gfCNCPoint1[24009] = {X 25.7631, Y 5.7856, Z -2.1667, A 0.000, B 0.000, C 0.000 }
gfCNCPoint1[24010] = {X 27.5759, Y 7.0515, Z -2.1667, A 0.000, B 0.000, C 0.000 }
gfCNCPoint1[24011] = {X 28.5579, Y 7.8754, Z -2.1667, A 0.000, B 0.000, C 0.000 }
gfCNCPoint1[24012] = {X 29.4785, Y 8.7676, Z -2.1667, A 0.000, B 0.000, C 0.000 }
gfCNCPoint1[24013] = {X 30.6864, Y 10.1626, Z -2.1667, A 0.000, B 0.000, C 0.000 }
gfCNCPoint1[24014] = {X 31.7443, Y 11.6745, Z -2.1667, A 0.000, B 0.000, C 0.000 }
gfCNCPoint1[24015] = {X 32.6409, Y 13.2874, Z -2.1667, A 0.000, B 0.000, C 0.000 }
gfCNCPoint1[24016] = {X 33.3666, Y 14.9840, Z -2.1667, A 0.000, B 0.000, C 0.000 }
gfCNCPoint1[24017] = {X 33.9177, Y 16.8152, Z -2.1667, A 0.000, B 0.000, C 0.000 }
gfCNCPoint1[24018] = {X 34.2900, Y 18.6910, Z -2.1667, A 0.000, B 0.000, C 0.000 }
gfCNCPoint1[24019] = {X 34.4801, Y 20.5940, Z -2.1667, A 0.000, B 0.000, C 0.000 }
gfCNCPoint1[24020] = {X 34.4863, Y 22.5063, Z -2.1667, A 0.000, B 0.000, C 0.000 }
gfCNCPoint1[24021] = {X 34.3084, Y 24.4105, Z -2.1667, A 0.000, B 0.000, C 0.000 }
gfCNCPoint1[24022] = {X 33.9482, Y 26.2886, Z -2.1667, A 0.000, B 0.000, C 0.000 }
gfCNCPoint1[24023] = {X 33.4648, Y 27.9398, Z -2.1667, A 0.000, B 0.000, C 0.000 }
gfCNCPoint1[24024] = {X 32.8126, Y 29.5319, Z -2.1667, A 0.000, B 0.000, C 0.000 }
gfCNCPoint1[24025] = {X 31.9989, Y 31.0478, Z -2.1667, A 0.000, B 0.000, C 0.000 }
gfCNCPoint1[24026] = {X 32.1285, Y 31.2838, Z -2.1667, A 0.000, B 0.000, C 0.000 }
gfCNCPoint1[24027] = {X 32.2512, Y 31.5235, Z -2.1667, A 0.000, B 0.000, C 0.000 }
gfCNCPoint1[24028] = {X 35.3025, Y 37.8269, Z -2.1667, A 0.000, B 0.000, C 0.000 }
gfCNCPoint1[24029] = {X 35.7263, Y 38.8573, Z -2.1667, A 0.000, B 0.000, C 0.000 }
gfCNCPoint1[24030] = {X 36.0224, Y 39.9313, Z -2.1667, A 0.000, B 0.000, C 0.000 }
gfCNCPoint1[24031] = {X 36.1865, Y 41.0332, Z -2.1667, A 0.000, B 0.000, C 0.000 }
gfCNCPoint1[24032] = {X 36.2163, Y 42.1469, Z -2.1667, A 0.000, B 0.000, C 0.000 }
gfCNCPoint1[24033] = {X 36.6306, Y 41.4259, Z -2.1667, A 0.000, B 0.000, C 0.000 }
gfCNCPoint1[24034] = {X 37.1613, Y 40.7857, Z -2.1667, A 0.000, B 0.000, C 0.000 }
gfCNCPoint1[24035] = {X 37.7930, Y 40.2449, Z -2.1667, A 0.000, B 0.000, C 0.000 }
gfCNCPoint1[24036] = {X 38.5073, Y 39.8191, Z -2.1667, A 0.000, B 0.000, C 0.000 }
gfCNCPoint1[24037] = {X 39.0456, Y 38.5336, Z -2.1667, A 0.000, B 0.000, C 0.000 }
gfCNCPoint1[24038] = {X 39.5416, Y 37.2312, Z -2.1667, A 0.000, B 0.000, C 0.000 }
gfCNCPoint1[24039] = {X 47.6703, Y 15.4045, Z -2.1667, A 0.000, B 0.000, C 0.000 }
gfCNCPoint1[24040] = {X 47.3200, Y 14.6512, Z -2.1667, A 0.000, B 0.000, C 0.000 }
gfCNCPoint1[24041] = {X 47.1026, Y 13.8493, Z -2.1667, A 0.000, B 0.000, C 0.000 }
gfCNCPoint1[24042] = {X 47.0244, Y 13.0222, Z -2.1667, A 0.000, B 0.000, C 0.000 }
gfCNCPoint1[24043] = {X 47.0242, Y 12.1868, Z -2.1667, A 0.000, B 0.000, C 0.000 }
gfCNCPoint1[24044] = {X 47.0722, Y 11.5041, Z -2.1667, A 0.000, B 0.000, C 0.000 }
gfCNCPoint1[24045] = {X 47.2152, Y 10.8349, Z -2.1667, A 0.000, B 0.000, C 0.000 }
gfCNCPoint1[24046] = {X 42.6031, Y 9.5051, Z -2.1667, A 0.000, B 0.000, C 0.000 }
gfCNCPoint1[24047] = {X 36.0439, Y 9.5051, Z -2.1667, A 0.000, B 0.000, C 0.000 }
gfCNCPoint1[24048] = {X 37.0532, Y 11.3861, Z -2.1667, A 0.000, B 0.000, C 0.000 }
gfCNCPoint1[24049] = {X 37.8813, Y 13.3537, Z -2.1667, A 0.000, B 0.000, C 0.000 }
gfCNCPoint1[24050] = {X 38.5455, Y 15.5364, Z -2.1667, A 0.000, B 0.000, C 0.000 }
gfCNCPoint1[24051] = {X 39.0050, Y 17.7712, Z -2.1667, A 0.000, B 0.000, C 0.000 }
gfCNCPoint1[24052] = {X 39.2560, Y 20.0389, Z -2.1667, A 0.000, B 0.000, C 0.000 }
gfCNCPoint1[24053] = {X 39.2962, Y 22.3201, Z -2.1667, A 0.000, B 0.000, C 0.000 }
gfCNCPoint1[24054] = {X 39.1255, Y 24.5952, Z -2.1667, A 0.000, B 0.000, C 0.000 }
gfCNCPoint1[24055] = {X 42.5394, Y 15.4281, Z -2.1667, A 0.000, B 0.000, C 0.000 }
gfCNCPoint1[24056] = {X 42.3081, Y 14.2498, Z -2.1667, A 0.000, B 0.000, C 0.000 }
gfCNCPoint1[24057] = {X 42.2245, Y 13.0519, Z -2.1667, A 0.000, B 0.000, C 0.000 }
gfCNCPoint1[24058] = {X 42.2242, Y 12.1868, Z -2.1667, A 0.000, B 0.000, C 0.000 }
gfCNCPoint1[24059] = {X 42.3194, Y 10.8326, Z -2.1667, A 0.000, B 0.000, C 0.000 }
gfCNCPoint1[24060] = {X 42.6031, Y 9.5051, Z -2.1667, A 0.000, B 0.000, C 0.000 }
gfCNCPoint1[24061] = {X 44.9092, Y 10.1700, Z -2.1667, A 0.000, B 0.000, C 0.000 }
gfCNCPoint1[24062] = {X 45.3323, Y 9.0551, Z -2.1667, A 0.000, B 0.000, C 0.000 }
gfCNCPoint1[24063] = {X 45.9317, Y 8.0242, Z -2.1667, A 0.000, B 0.000, C 0.000 }
gfCNCPoint1[24064] = {X 46.6913, Y 7.1051, Z -2.1667, A 0.000, B 0.000, C 0.000 }
gfCNCPoint1[24065] = {X 31.2094, Y 7.1051, Z -2.1667, A 0.000, B 0.000, C 0.000 }
gfCNCPoint1[24066] = {X 32.2249, Y 8.2452, Z -2.1667, A 0.000, B 0.000, C 0.000 }
gfCNCPoint1[24067] = {X 33.1518, Y 9.4585, Z -2.1667, A 0.000, B 0.000, C 0.000 }
gfCNCPoint1[24068] = {X 33.9848, Y 10.7380, Z -2.1667, A 0.000, B 0.000, C 0.000 }
gfCNCPoint1[24069] = {X 34.8849, Y 12.4149, Z -2.1667, A 0.000, B 0.000, C 0.000 }
gfCNCPoint1[24070] = {X 35.6240, Y 14.1688, Z -2.1667, A 0.000, B 0.000, C 0.000 }
gfCNCPoint1[24071] = {X 36.2218, Y 16.1371, Z -2.1667, A 0.000, B 0.000, C 0.000 }
gfCNCPoint1[24072] = {X 36.6354, Y 18.1522, Z -2.1667, A 0.000, B 0.000, C 0.000 }
gfCNCPoint1[24073] = {X 36.8612, Y 20.1969, Z -2.1667, A 0.000, B 0.000, C 0.000 }
gfCNCPoint1[24074] = {X 36.8971, Y 22.2537, Z -2.1667, A 0.000, B 0.000, C 0.000 }
gfCNCPoint1[24075] = {X 36.7431, Y 24.3050, Z -2.1667, A 0.000, B 0.000, C 0.000 }
gfCNCPoint1[24076] = {X 36.5495, Y 25.5833, Z -2.1667, A 0.000, B 0.000, C 0.000 }
gfCNCPoint1[24077] = {X 36.2821, Y 26.8481, Z -2.1667, A 0.000, B 0.000, C 0.000 }
gfCNCPoint1[24078] = {X 35.8735, Y 28.3068, Z -2.1667, A 0.000, B 0.000, C 0.000 }
gfCNCPoint1[24079] = {X 35.3497, Y 29.7282, Z -2.1667, A 0.000, B 0.000, C 0.000 }
gfCNCPoint1[24080] = {X 34.7142, Y 31.1033, Z -2.1667, A 0.000, B 0.000, C 0.000 }
gfCNCPoint1[24081] = {X 37.2850, Y 36.4140, Z -2.1667, A 0.000, B 0.000, C 0.000 }
gfCNCPoint1[24082] = {X 45.0744, Y 15.4982, Z -2.1667, A 0.000, B 0.000, C 0.000 }
gfCNCPoint1[24083] = {X 44.7426, Y 14.2853, Z -2.1667, A 0.000, B 0.000, C 0.000 }
gfCNCPoint1[24084] = {X 44.6244, Y 13.0334, Z -2.1667, A 0.000, B 0.000, C 0.000 }
gfCNCPoint1[24085] = {X 44.6242, Y 12.1868, Z -2.1667, A 0.000, B 0.000, C 0.000 }
gfCNCPoint1[24086] = {X 44.6958, Y 11.1684, Z -2.1667, A 0.000, B 0.000, C 0.000 }
gfCNCPoint1[24087] = {X 44.9092, Y 10.1700, Z -2.1667, A 0.000, B 0.000, C 0.000 }
gfCNCPoint1[24088] = {X 47.2152, Y 10.8349, Z -2.1667, A 0.000, B 0.000, C 0.000 }
gfCNCPoint1[24089] = {X 47.4988, Y 10.0875, Z -2.1667, A 0.000, B 0.000, C 0.000 }
gfCNCPoint1[24090] = {X 47.9006, Y 9.3965, Z -2.1667, A 0.000, B 0.000, C 0.000 }
gfCNCPoint1[24091] = {X 48.4099, Y 8.7804, Z -2.1667, A 0.000, B 0.000, C 0.000 }
gfCNCPoint1[24092] = {X 49.1544, Y 8.1553, Z -2.1667, A 0.000, B 0.000, C 0.000 }
gfCNCPoint1[24093] = {X 50.0080, Y 7.6903, Z -2.1667, A 0.000, B 0.000, C 0.000 }
gfCNCPoint1[24094] = {X 50.9369, Y 7.4036, Z -2.1667, A 0.000, B 0.000, C 0.000 }
gfCNCPoint1[24095] = {X 51.9042, Y 7.3068, Z -2.1667, A 0.000, B 0.000, C 0.000 }
gfCNCPoint1[24096] = {X 59.6221, Y 7.3068, Z -2.1667, A 0.000, B 0.000, C 0.000 }
gfCNCPoint1[24097] = {X 60.5894, Y 7.4036, Z -2.1667, A 0.000, B 0.000, C 0.000 }
gfCNCPoint1[24098] = {X 61.5183, Y 7.6903, Z -2.1667, A 0.000, B 0.000, C 0.000 }
gfCNCPoint1[24099] = {X 62.3720, Y 8.1553, Z -2.1667, A 0.000, B 0.000, C 0.000 }
gfCNCPoint1[24100] = {X 63.1165, Y 8.7804, Z -2.1667, A 0.000, B 0.000, C 0.000 }
gfCNCPoint1[24101] = {X 63.7054, Y 9.5145, Z -2.1667, A 0.000, B 0.000, C 0.000 }
gfCNCPoint1[24102] = {X 64.1425, Y 10.3481, Z -2.1667, A 0.000, B 0.000, C 0.000 }
gfCNCPoint1[24103] = {X 64.4114, Y 11.2500, Z -2.1667, A 0.000, B 0.000, C 0.000 }
gfCNCPoint1[24104] = {X 64.5021, Y 12.1868, Z -2.1667, A 0.000, B 0.000, C 0.000 }
gfCNCPoint1[24105] = {X 64.5019, Y 13.0237, Z -2.1667, A 0.000, B 0.000, C 0.000 }
gfCNCPoint1[24106] = {X 64.4204, Y 13.8671, Z -2.1667, A 0.000, B 0.000, C 0.000 }
gfCNCPoint1[24107] = {X 64.1943, Y 14.6838, Z -2.1667, A 0.000, B 0.000, C 0.000 }
gfCNCPoint1[24108] = {X 63.8303, Y 15.4490, Z -2.1667, A 0.000, B 0.000, C 0.000 }
gfCNCPoint1[24109] = {X 63.9941, Y 15.8770, Z -2.1667, A 0.000, B 0.000, C 0.000 }
gfCNCPoint1[24110] = {X 72.9532, Y 39.8573, Z -2.1667, A 0.000, B 0.000, C 0.000 }
gfCNCPoint1[24111] = {X 73.8435, Y 40.4391, Z -2.1667, A 0.000, B 0.000, C 0.000 }
gfCNCPoint1[24112] = {X 74.5866, Y 41.2001, Z -2.1667, A 0.000, B 0.000, C 0.000 }
gfCNCPoint1[24113] = {X 75.1472, Y 42.1040, Z -2.1667, A 0.000, B 0.000, C 0.000 }
gfCNCPoint1[24114] = {X 75.4987, Y 43.1079, Z -2.1667, A 0.000, B 0.000, C 0.000 }
gfCNCPoint1[24115] = {X 75.6243, Y 44.1640, Z -2.1667, A 0.000, B 0.000, C 0.000 }
gfCNCPoint1[24116] = {X 75.6245, Y 45.0000, Z -2.1667, A 0.000, B 0.000, C 0.000 }
gfCNCPoint1[24117] = {X 75.5307, Y 45.9520, Z -2.1667, A 0.000, B 0.000, C 0.000 }
gfCNCPoint1[24118] = {X 75.2530, Y 46.8675, Z -2.1667, A 0.000, B 0.000, C 0.000 }
gfCNCPoint1[24119] = {X 74.8020, Y 47.7112, Z -2.1667, A 0.000, B 0.000, C 0.000 }
gfCNCPoint1[24120] = {X 74.1951, Y 48.4507, Z -2.1667, A 0.000, B 0.000, C 0.000 }
gfCNCPoint1[24121] = {X 73.4556, Y 49.0576, Z -2.1667, A 0.000, B 0.000, C 0.000 }
gfCNCPoint1[24122] = {X 72.6120, Y 49.5085, Z -2.1667, A 0.000, B 0.000, C 0.000 }
gfCNCPoint1[24123] = {X 71.6965, Y 49.7862, Z -2.1667, A 0.000, B 0.000, C 0.000 }
gfCNCPoint1[24124] = {X 70.7445, Y 49.8800, Z -2.1667, A 0.000, B 0.000, C 0.000 }
gfCNCPoint1[24125] = {X 64.1851, Y 49.8800, Z -2.1667, A 0.000, B 0.000, C 0.000 }
gfCNCPoint1[24126] = {X 63.2331, Y 49.7862, Z -2.1667, A 0.000, B 0.000, C 0.000 }
gfCNCPoint1[24127] = {X 62.3176, Y 49.5085, Z -2.1667, A 0.000, B 0.000, C 0.000 }
gfCNCPoint1[24128] = {X 61.4740, Y 49.0576, Z -2.1667, A 0.000, B 0.000, C 0.000 }
gfCNCPoint1[24129] = {X 60.7345, Y 48.4507, Z -2.1667, A 0.000, B 0.000, C 0.000 }
gfCNCPoint1[24130] = {X 60.1276, Y 47.7112, Z -2.1667, A 0.000, B 0.000, C 0.000 }
gfCNCPoint1[24131] = {X 59.6766, Y 46.8675, Z -2.1667, A 0.000, B 0.000, C 0.000 }
gfCNCPoint1[24132] = {X 59.3989, Y 45.9520, Z -2.1667, A 0.000, B 0.000, C 0.000 }
gfCNCPoint1[24133] = {X 59.3051, Y 45.0000, Z -2.1667, A 0.000, B 0.000, C 0.000 }
gfCNCPoint1[24134] = {X 59.3052, Y 44.2029, Z -2.1667, A 0.000, B 0.000, C 0.000 }
gfCNCPoint1[24135] = {X 59.3848, Y 43.3308, Z -2.1667, A 0.000, B 0.000, C 0.000 }
gfCNCPoint1[24136] = {X 59.6190, Y 42.4870, Z -2.1667, A 0.000, B 0.000, C 0.000 }
gfCNCPoint1[24137] = {X 60.0003, Y 41.6986, Z -2.1667, A 0.000, B 0.000, C 0.000 }
gfCNCPoint1[24138] = {X 59.6160, Y 40.6492, Z -2.1667, A 0.000, B 0.000, C 0.000 }
gfCNCPoint1[24139] = {X 52.4655, Y 40.6492, Z -2.1667, A 0.000, B 0.000, C 0.000 }
gfCNCPoint1[24140] = {X 51.9464, Y 42.0438, Z -2.1667, A 0.000, B 0.000, C 0.000 }
gfCNCPoint1[24141] = {X 52.2214, Y 42.7234, Z -2.1667, A 0.000, B 0.000, C 0.000 }
gfCNCPoint1[24142] = {X 52.3914, Y 43.4366, Z -2.1667, A 0.000, B 0.000, C 0.000 }
gfCNCPoint1[24143] = {X 52.4528, Y 44.1672, Z -2.1667, A 0.000, B 0.000, C 0.000 }
gfCNCPoint1[24144] = {X 52.4529, Y 45.0000, Z -2.1667, A 0.000, B 0.000, C 0.000 }
gfCNCPoint1[24145] = {X 52.3592, Y 45.9520, Z -2.1667, A 0.000, B 0.000, C 0.000 }
gfCNCPoint1[24146] = {X 52.0815, Y 46.8675, Z -2.1667, A 0.000, B 0.000, C 0.000 }
gfCNCPoint1[24147] = {X 51.6305, Y 47.7112, Z -2.1667, A 0.000, B 0.000, C 0.000 }
gfCNCPoint1[24148] = {X 51.0236, Y 48.4507, Z -2.1667, A 0.000, B 0.000, C 0.000 }
gfCNCPoint1[24149] = {X 50.2841, Y 49.0576, Z -2.1667, A 0.000, B 0.000, C 0.000 }
gfCNCPoint1[24150] = {X 49.4404, Y 49.5085, Z -2.1667, A 0.000, B 0.000, C 0.000 }
gfCNCPoint1[24151] = {X 48.5250, Y 49.7862, Z -2.1667, A 0.000, B 0.000, C 0.000 }
gfCNCPoint1[24152] = {X 47.5729, Y 49.8800, Z -2.1667, A 0.000, B 0.000, C 0.000 }
gfCNCPoint1[24153] = {X 40.6393, Y 49.8800, Z -2.1667, A 0.000, B 0.000, C 0.000 }
gfCNCPoint1[24154] = {X 39.6433, Y 49.7773, Z -2.1667, A 0.000, B 0.000, C 0.000 }
gfCNCPoint1[24155] = {X 38.6892, Y 49.4734, Z -2.1667, A 0.000, B 0.000, C 0.000 }
gfCNCPoint1[24156] = {X 37.8173, Y 48.9813, Z -2.1667, A 0.000, B 0.000, C 0.000 }
gfCNCPoint1[24157] = {X 37.0641, Y 48.3215, Z -2.1667, A 0.000, B 0.000, C 0.000 }
gfCNCPoint1[24158] = {X 36.5085, Y 47.5983, Z -2.1667, A 0.000, B 0.000, C 0.000 }
gfCNCPoint1[24159] = {X 36.0972, Y 46.7843, Z -2.1667, A 0.000, B 0.000, C 0.000 }
gfCNCPoint1[24160] = {X 35.8445, Y 45.9080, Z -2.1667, A 0.000, B 0.000, C 0.000 }
gfCNCPoint1[24161] = {X 35.7593, Y 45.0000, Z -2.1667, A 0.000, B 0.000, C 0.000 }
gfCNCPoint1[24162] = {X 35.7593, Y 44.7148, Z -2.1667, A 0.000, B 0.000, C 0.000 }
gfCNCPoint1[24163] = {X 36.2393, Y 44.7148, Z -2.1667, A 0.000, B 0.000, C 0.000 }
gfCNCPoint1[24164] = {X 36.2397, Y 44.1483, Z -2.1667, A 0.000, B 0.000, C 0.000 }
gfCNCPoint1[24165] = {X 36.3681, Y 43.1519, Z -2.1667, A 0.000, B 0.000, C 0.000 }
gfCNCPoint1[24166] = {X 36.7192, Y 42.2107, Z -2.1667, A 0.000, B 0.000, C 0.000 }
gfCNCPoint1[24167] = {X 37.2745, Y 41.3736, Z -2.1667, A 0.000, B 0.000, C 0.000 }
gfCNCPoint1[24168] = {X 38.0053, Y 40.6843, Z -2.1667, A 0.000, B 0.000, C 0.000 }
gfCNCPoint1[24169] = {X 38.8734, Y 40.1787, Z -2.1667, A 0.000, B 0.000, C 0.000 }
gfCNCPoint1[24170] = {X 39.4565, Y 38.7984, Z -2.1667, A 0.000, B 0.000, C 0.000 }
gfCNCPoint1[24171] = {X 39.9914, Y 37.3987, Z -2.1667, A 0.000, B 0.000, C 0.000 }
gfCNCPoint1[24172] = {X 48.2011, Y 15.3544, Z -2.1667, A 0.000, B 0.000, C 0.000 }
gfCNCPoint1[24173] = {X 47.8187, Y 14.6115, Z -2.1667, A 0.000, B 0.000, C 0.000 }
gfCNCPoint1[24174] = {X 47.5835, Y 13.8097, Z -2.1667, A 0.000, B 0.000, C 0.000 }
gfCNCPoint1[24175] = {X 47.5042, Y 12.9779, Z -2.1667, A 0.000, B 0.000, C 0.000 }
gfCNCPoint1[24176] = {X 47.5042, Y 12.1868, Z -2.1667, A 0.000, B 0.000, C 0.000 }
gfCNCPoint1[24177] = {X 47.6145, Y 11.2077, Z -2.1667, A 0.000, B 0.000, C 0.000 }
gfCNCPoint1[24178] = {X 47.9400, Y 10.2777, Z -2.1667, A 0.000, B 0.000, C 0.000 }
gfCNCPoint1[24179] = {X 48.4642, Y 9.4435, Z -2.1667, A 0.000, B 0.000, C 0.000 }
gfCNCPoint1[24180] = {X 49.1609, Y 8.7468, Z -2.1667, A 0.000, B 0.000, C 0.000 }
gfCNCPoint1[24181] = {X 49.9951, Y 8.2226, Z -2.1667, A 0.000, B 0.000, C 0.000 }
gfCNCPoint1[24182] = {X 50.9251, Y 7.8971, Z -2.1667, A 0.000, B 0.000, C 0.000 }
gfCNCPoint1[24183] = {X 51.9042, Y 7.7868, Z -2.1667, A 0.000, B 0.000, C 0.000 }
gfCNCPoint1[24184] = {X 59.6221, Y 7.7868, Z -2.1667, A 0.000, B 0.000, C 0.000 }
gfCNCPoint1[24185] = {X 60.6012, Y 7.8971, Z -2.1667, A 0.000, B 0.000, C 0.000 }
gfCNCPoint1[24186] = {X 61.5312, Y 8.2226, Z -2.1667, A 0.000, B 0.000, C 0.000 }
gfCNCPoint1[24187] = {X 62.3655, Y 8.7468, Z -2.1667, A 0.000, B 0.000, C 0.000 }
gfCNCPoint1[24188] = {X 63.0622, Y 9.4435, Z -2.1667, A 0.000, B 0.000, C 0.000 }
gfCNCPoint1[24189] = {X 63.5864, Y 10.2777, Z -2.1667, A 0.000, B 0.000, C 0.000 }
gfCNCPoint1[24190] = {X 63.9118, Y 11.2077, Z -2.1667, A 0.000, B 0.000, C 0.000 }
gfCNCPoint1[24191] = {X 64.0221, Y 12.1868, Z -2.1667, A 0.000, B 0.000, C 0.000 }
gfCNCPoint1[24192] = {X 64.0219, Y 13.0233, Z -2.1667, A 0.000, B 0.000, C 0.000 }
gfCNCPoint1[24193] = {X 63.9336, Y 13.8564, Z -2.1667, A 0.000, B 0.000, C 0.000 }
gfCNCPoint1[24194] = {X 63.6889, Y 14.6576, Z -2.1667, A 0.000, B 0.000, C 0.000 }
gfCNCPoint1[24195] = {X 63.2969, Y 15.3980, Z -2.1667, A 0.000, B 0.000, C 0.000 }
gfCNCPoint1[24196] = {X 63.5448, Y 16.0461, Z -2.1667, A 0.000, B 0.000, C 0.000 }
gfCNCPoint1[24197] = {X 66.1094, Y 22.8602, Z -2.1667, A 0.000, B 0.000, C 0.000 }
gfCNCPoint1[24198] = {X 72.2834, Y 39.4716, Z -2.1667, A 0.000, B 0.000, C 0.000 }
gfCNCPoint1[24199] = {X 72.5762, Y 40.2082, Z -2.1667, A 0.000, B 0.000, C 0.000 }
gfCNCPoint1[24200] = {X 73.4340, Y 40.7265, Z -2.1667, A 0.000, B 0.000, C 0.000 }
gfCNCPoint1[24201] = {X 74.1523, Y 41.4256, Z -2.1667, A 0.000, B 0.000, C 0.000 }
gfCNCPoint1[24202] = {X 74.6938, Y 42.2690, Z -2.1667, A 0.000, B 0.000, C 0.000 }
gfCNCPoint1[24203] = {X 75.0303, Y 43.2131, Z -2.1667, A 0.000, B 0.000, C 0.000 }
gfCNCPoint1[24204] = {X 75.1445, Y 44.2089, Z -2.1667, A 0.000, B 0.000, C 0.000 }
gfCNCPoint1[24205] = {X 75.1445, Y 45.0000, Z -2.1667, A 0.000, B 0.000, C 0.000 }
gfCNCPoint1[24206] = {X 75.0341, Y 45.9791, Z -2.1667, A 0.000, B 0.000, C 0.000 }
gfCNCPoint1[24207] = {X 74.7087, Y 46.9091, Z -2.1667, A 0.000, B 0.000, C 0.000 }
gfCNCPoint1[24208] = {X 74.1845, Y 47.7434, Z -2.1667, A 0.000, B 0.000, C 0.000 }
gfCNCPoint1[24209] = {X 73.4878, Y 48.4401, Z -2.1667, A 0.000, B 0.000, C 0.000 }
gfCNCPoint1[24210] = {X 72.6535, Y 48.9643, Z -2.1667, A 0.000, B 0.000, C 0.000 }
gfCNCPoint1[24211] = {X 71.7236, Y 49.2897, Z -2.1667, A 0.000, B 0.000, C 0.000 }
gfCNCPoint1[24212] = {X 70.7445, Y 49.4000, Z -2.1667, A 0.000, B 0.000, C 0.000 }
gfCNCPoint1[24213] = {X 64.1851, Y 49.4000, Z -2.1667, A 0.000, B 0.000, C 0.000 }
gfCNCPoint1[24214] = {X 63.2060, Y 49.2897, Z -2.1667, A 0.000, B 0.000, C 0.000 }
gfCNCPoint1[24215] = {X 62.2760, Y 48.9643, Z -2.1667, A 0.000, B 0.000, C 0.000 }
gfCNCPoint1[24216] = {X 61.4418, Y 48.4401, Z -2.1667, A 0.000, B 0.000, C 0.000 }
gfCNCPoint1[24217] = {X 60.7451, Y 47.7434, Z -2.1667, A 0.000, B 0.000, C 0.000 }
gfCNCPoint1[24218] = {X 60.2209, Y 46.9091, Z -2.1667, A 0.000, B 0.000, C 0.000 }
gfCNCPoint1[24219] = {X 59.8955, Y 45.9791, Z -2.1667, A 0.000, B 0.000, C 0.000 }
gfCNCPoint1[24220] = {X 59.7851, Y 45.0000, Z -2.1667, A 0.000, B 0.000, C 0.000 }
gfCNCPoint1[24221] = {X 59.7856, Y 44.1483, Z -2.1667, A 0.000, B 0.000, C 0.000 }
gfCNCPoint1[24222] = {X 59.8784, Y 43.3075, Z -2.1667, A 0.000, B 0.000, C 0.000 }
gfCNCPoint1[24223] = {X 60.1305, Y 42.5001, Z -2.1667, A 0.000, B 0.000, C 0.000 }
gfCNCPoint1[24224] = {X 60.5324, Y 41.7558, Z -2.1667, A 0.000, B 0.000, C 0.000 }
gfCNCPoint1[24225] = {X 59.9515, Y 40.1692, Z -2.1667, A 0.000, B 0.000, C 0.000 }
gfCNCPoint1[24226] = {X 52.1320, Y 40.1692, Z -2.1667, A 0.000, B 0.000, C 0.000 }
gfCNCPoint1[24227] = {X 51.4219, Y 42.0768, Z -2.1667, A 0.000, B 0.000, C 0.000 }
gfCNCPoint1[24228] = {X 51.7251, Y 42.7530, Z -2.1667, A 0.000, B 0.000, C 0.000 }
gfCNCPoint1[24229] = {X 51.9105, Y 43.4705, Z -2.1667, A 0.000, B 0.000, C 0.000 }
gfCNCPoint1[24230] = {X 51.9729, Y 44.2089, Z -2.1667, A 0.000, B 0.000, C 0.000 }
gfCNCPoint1[24231] = {X 51.9729, Y 45.0000, Z -2.1667, A 0.000, B 0.000, C 0.000 }
gfCNCPoint1[24232] = {X 51.8626, Y 45.9791, Z -2.1667, A 0.000, B 0.000, C 0.000 }
gfCNCPoint1[24233] = {X 51.5372, Y 46.9091, Z -2.1667, A 0.000, B 0.000, C 0.000 }
gfCNCPoint1[24234] = {X 51.0130, Y 47.7434, Z -2.1667, A 0.000, B 0.000, C 0.000 }
gfCNCPoint1[24235] = {X 50.3163, Y 48.4401, Z -2.1667, A 0.000, B 0.000, C 0.000 }
gfCNCPoint1[24236] = {X 49.4820, Y 48.9643, Z -2.1667, A 0.000, B 0.000, C 0.000 }
gfCNCPoint1[24237] = {X 48.5520, Y 49.2897, Z -2.1667, A 0.000, B 0.000, C 0.000 }
gfCNCPoint1[24238] = {X 47.5729, Y 49.4000, Z -2.1667, A 0.000, B 0.000, C 0.000 }
gfCNCPoint1[24239] = {X 40.6393, Y 49.4000, Z -2.1667, A 0.000, B 0.000, C 0.000 }
gfCNCPoint1[24240] = {X 39.6602, Y 49.2897, Z -2.1667, A 0.000, B 0.000, C 0.000 }
gfCNCPoint1[24241] = {X 38.7302, Y 48.9643, Z -2.1667, A 0.000, B 0.000, C 0.000 }
gfCNCPoint1[24242] = {X 37.8959, Y 48.4401, Z -2.1667, A 0.000, B 0.000, C 0.000 }
gfCNCPoint1[24243] = {X 37.1992, Y 47.7434, Z -2.1667, A 0.000, B 0.000, C 0.000 }
gfCNCPoint1[24244] = {X 36.6750, Y 46.9091, Z -2.1667, A 0.000, B 0.000, C 0.000 }
gfCNCPoint1[24245] = {X 36.3496, Y 45.9791, Z -2.1667, A 0.000, B 0.000, C 0.000 }
gfCNCPoint1[24246] = {X 36.2393, Y 45.0000, Z -2.1667, A 0.000, B 0.000, C 0.000 }
gfCNCPoint1[24247] = {X 36.2393, Y 44.7148, Z -2.1667, A 0.000, B 0.000, C 0.000 }
gfCNCPoint1[24248] = {X 35.7593, Y 44.7148, Z -2.1667, A 0.000, B 0.000, C 0.000 }
gfCNCPoint1[24249] = {X 35.2211, Y 46.0074, Z -2.1667, A 0.000, B 0.000, C 0.000 }
gfCNCPoint1[24250] = {X 34.4930, Y 47.2034, Z -2.1667, A 0.000, B 0.000, C 0.000 }
gfCNCPoint1[24251] = {X 33.5918, Y 48.2750, Z -2.1667, A 0.000, B 0.000, C 0.000 }
gfCNCPoint1[24252] = {X 33.2092, Y 48.6435, Z -2.1667, A 0.000, B 0.000, C 0.000 }
gfCNCPoint1[24253] = {X 32.8060, Y 48.9892, Z -2.1667, A 0.000, B 0.000, C 0.000 }
gfCNCPoint1[24254] = {X 32.2647, Y 49.4269, Z -2.1667, A 0.000, B 0.000, C 0.000 }
gfCNCPoint1[24255] = {X 31.1788, Y 50.1808, Z -2.1667, A 0.000, B 0.000, C 0.000 }
gfCNCPoint1[24256] = {X 29.9962, Y 50.7716, Z -2.1667, A 0.000, B 0.000, C 0.000 }
gfCNCPoint1[24257] = {X 28.7413, Y 51.1872, Z -2.1667, A 0.000, B 0.000, C 0.000 }
gfCNCPoint1[24258] = {X 27.4399, Y 51.4190, Z -2.1667, A 0.000, B 0.000, C 0.000 }
gfCNCPoint1[24259] = {X 26.1186, Y 51.4622, Z -2.1667, A 0.000, B 0.000, C 0.000 }
gfCNCPoint1[24260] = {X 24.2349, Y 52.3474, Z -2.1667, A 0.000, B 0.000, C 0.000 }
gfCNCPoint1[24261] = {X 22.2997, Y 53.1135, Z -2.1667, A 0.000, B 0.000, C 0.000 }
gfCNCPoint1[24262] = {X 20.3206, Y 53.7576, Z -2.1667, A 0.000, B 0.000, C 0.000 }
gfCNCPoint1[24263] = {X 18.2342, Y 54.2907, Z -2.1667, A 0.000, B 0.000, C 0.000 }
gfCNCPoint1[24264] = {X 16.1125, Y 54.6590, Z -2.1667, A 0.000, B 0.000, C 0.000 }
gfCNCPoint1[24265] = {X 13.9685, Y 54.8603, Z -2.1667, A 0.000, B 0.000, C 0.000 }
gfCNCPoint1[24266] = {X 11.8153, Y 54.8932, Z -2.1667, A 0.000, B 0.000, C 0.000 }
gfCNCPoint1[24267] = {X 9.6662, Y 54.7576, Z -2.1667, A 0.000, B 0.000, C 0.000 }
gfCNCPoint1[24268] = {X 7.5342, Y 54.4544, Z -2.1667, A 0.000, B 0.000, C 0.000 }
gfCNCPoint1[24269] = {X 7.4442, Y 54.4378, Z -2.1667, A 0.000, B 0.000, C 0.000 }
gfCNCPoint1[24270] = {X 7.3543, Y 54.4209, Z -2.1667, A 0.000, B 0.000, C 0.000 }
gfCNCPoint1[24271] = {X 6.0186, Y 54.1320, Z -2.1667, A 0.000, B 0.000, C 0.000 }
gfCNCPoint1[24272] = {X 4.7035, Y 53.7608, Z -2.1667, A 0.000, B 0.000, C 0.000 }
gfCNCPoint1[24273] = {X 4.7035, Y 95.2949, Z -2.1667, A 0.000, B 0.000, C 0.000 }
gfCNCPoint1[24274] = {X 117.9387, Y 95.2949, Z -2.1667, A 0.000, B 0.000, C 0.000 }
gfCNCPoint1[24275] = {X 118.3618, Y 94.0772, Z -2.1667, A 0.000, B 0.000, C 0.000 }
gfCNCPoint1[24276] = {X 118.9931, Y 92.9531, Z -2.1667, A 0.000, B 0.000, C 0.000 }
gfCNCPoint1[24277] = {X 119.8127, Y 91.9580, Z -2.1667, A 0.000, B 0.000, C 0.000 }
gfCNCPoint1[24278] = {X 120.7950, Y 91.1231, Z -2.1667, A 0.000, B 0.000, C 0.000 }
gfCNCPoint1[24279] = {X 121.9092, Y 90.4746, Z -2.1667, A 0.000, B 0.000, C 0.000 }
gfCNCPoint1[24280] = {X 123.1203, Y 90.0328, Z -2.1667, A 0.000, B 0.000, C 0.000 }
gfCNCPoint1[24281] = {X 124.3904, Y 89.8115, Z -2.1667, A 0.000, B 0.000, C 0.000 }
gfCNCPoint1[24282] = {X 125.0451, Y 89.7129, Z -2.1667, A 0.000, B 0.000, C 0.000 }
gfCNCPoint1[24283] = {X 125.3563, Y 89.6659, Z -2.1667, A 0.000, B 0.000, C 0.000 }
gfCNCPoint1[24284] = {X 125.6659, Y 89.6088, Z -2.1667, A 0.000, B 0.000, C 0.000 }
gfCNCPoint1[24285] = {X 126.4927, Y 88.7981, Z -2.1667, A 0.000, B 0.000, C 0.000 }
gfCNCPoint1[24286] = {X 127.2853, Y 87.9540, Z -2.1667, A 0.000, B 0.000, C 0.000 }
gfCNCPoint1[24287] = {X 152.2078, Y 60.5856, Z -2.1667, A 0.000, B 0.000, C 0.000 }
gfCNCPoint1[24288] = {X 152.0685, Y 59.7903, Z -2.1667, A 0.000, B 0.000, C 0.000 }
gfCNCPoint1[24289] = {X 152.0181, Y 58.9845, Z -2.1667, A 0.000, B 0.000, C 0.000 }
gfCNCPoint1[24290] = {X 152.0180, Y 58.0000, Z -2.1667, A 0.000, B 0.000, C 0.000 }
gfCNCPoint1[24291] = {X 152.1286, Y 56.7358, Z -2.1667, A 0.000, B 0.000, C 0.000 }
gfCNCPoint1[24292] = {X 152.4570, Y 55.5101, Z -2.1667, A 0.000, B 0.000, C 0.000 }
gfCNCPoint1[24293] = {X 152.9933, Y 54.3600, Z -2.1667, A 0.000, B 0.000, C 0.000 }
gfCNCPoint1[24294] = {X 153.7212, Y 53.3205, Z -2.1667, A 0.000, B 0.000, C 0.000 }
gfCNCPoint1[24295] = {X 154.6185, Y 52.4232, Z -2.1667, A 0.000, B 0.000, C 0.000 }
gfCNCPoint1[24296] = {X 155.6580, Y 51.6953, Z -2.1667, A 0.000, B 0.000, C 0.000 }
gfCNCPoint1[24297] = {X 156.8081, Y 51.1590, Z -2.1667, A 0.000, B 0.000, C 0.000 }
gfCNCPoint1[24298] = {X 158.0338, Y 50.8306, Z -2.1667, A 0.000, B 0.000, C 0.000 }
gfCNCPoint1[24299] = {X 159.2980, Y 50.7200, Z -2.1667, A 0.000, B 0.000, C 0.000 }
gfCNCPoint1[24300] = {X 178.5335, Y 50.7200, Z -2.1667, A 0.000, B 0.000, C 0.000 }
gfCNCPoint1[24301] = {X 179.7867, Y 50.8287, Z -2.1667, A 0.000, B 0.000, C 0.000 }
gfCNCPoint1[24302] = {X 181.0025, Y 51.1515, Z -2.1667, A 0.000, B 0.000, C 0.000 }
gfCNCPoint1[24303] = {X 182.1446, Y 51.6787, Z -2.1667, A 0.000, B 0.000, C 0.000 }
gfCNCPoint1[24304] = {X 183.1789, Y 52.3947, Z -2.1667, A 0.000, B 0.000, C 0.000 }
gfCNCPoint1[24305] = {X 184.0874, Y 53.2933, Z -2.1667, A 0.000, B 0.000, C 0.000 }
gfCNCPoint1[24306] = {X 184.8248, Y 54.3369, Z -2.1667, A 0.000, B 0.000, C 0.000 }
gfCNCPoint1[24307] = {X 185.3684, Y 55.4934, Z -2.1667, A 0.000, B 0.000, C 0.000 }
gfCNCPoint1[24308] = {X 185.7014, Y 56.7271, Z -2.1667, A 0.000, B 0.000, C 0.000 }
gfCNCPoint1[24309] = {X 185.8135, Y 58.0000, Z -2.1667, A 0.000, B 0.000, C 0.000 }
gfCNCPoint1[24310] = {X 185.8133, Y 58.9942, Z -2.1667, A 0.000, B 0.000, C 0.000 }
gfCNCPoint1[24311] = {X 185.7647, Y 59.7754, Z -2.1667, A 0.000, B 0.000, C 0.000 }
gfCNCPoint1[24312] = {X 185.6326, Y 60.5469, Z -2.1667, A 0.000, B 0.000, C 0.000 }
gfCNCPoint1[24313] = {X 211.6600, Y 88.9543, Z -2.1667, A 0.000, B 0.000, C 0.000 }
gfCNCPoint1[24314] = {X 212.0327, Y 89.3395, Z -2.1667, A 0.000, B 0.000, C 0.000 }
gfCNCPoint1[24315] = {X 212.4256, Y 89.7041, Z -2.1667, A 0.000, B 0.000, C 0.000 }
gfCNCPoint1[24316] = {X 212.6034, Y 89.7421, Z -2.1667, A 0.000, B 0.000, C 0.000 }
gfCNCPoint1[24317] = {X 213.4472, Y 89.8484, Z -2.1667, A 0.000, B 0.000, C 0.000 }
gfCNCPoint1[24318] = {X 214.4293, Y 89.7715, Z -2.1667, A 0.000, B 0.000, C 0.000 }
gfCNCPoint1[24319] = {X 215.4130, Y 89.7179, Z -2.1667, A 0.000, B 0.000, C 0.000 }
gfCNCPoint1[24320] = {X 215.6265, Y 89.6940, Z -2.1667, A 0.000, B 0.000, C 0.000 }
gfCNCPoint1[24321] = {X 215.8228, Y 89.6066, Z -2.1667, A 0.000, B 0.000, C 0.000 }
gfCNCPoint1[24322] = {X 239.3474, Y 74.5355, Z -2.1667, A 0.000, B 0.000, C 0.000 }
gfCNCPoint1[24323] = {X 220.5436, Y 67.1559, Z -2.1667, A 0.000, B 0.000, C 0.000 }
gfCNCPoint1[24324] = {X 219.0952, Y 66.6698, Z -2.1667, A 0.000, B 0.000, C 0.000 }
gfCNCPoint1[24325] = {X 217.6007, Y 66.3530, Z -2.1667, A 0.000, B 0.000, C 0.000 }
gfCNCPoint1[24326] = {X 216.0797, Y 66.2097, Z -2.1667, A 0.000, B 0.000, C 0.000 }
gfCNCPoint1[24327] = {X 214.8529, Y 66.0625, Z -2.1667, A 0.000, B 0.000, C 0.000 }
gfCNCPoint1[24328] = {X 213.6687, Y 65.7099, Z -2.1667, A 0.000, B 0.000, C 0.000 }
gfCNCPoint1[24329] = {X 212.5612, Y 65.1621, Z -2.1667, A 0.000, B 0.000, C 0.000 }
gfCNCPoint1[24330] = {X 211.5622, Y 64.4349, Z -2.1667, A 0.000, B 0.000, C 0.000 }
gfCNCPoint1[24331] = {X 210.7006, Y 63.5492, Z -2.1667, A 0.000, B 0.000, C 0.000 }
gfCNCPoint1[24332] = {X 210.0012, Y 62.5306, Z -2.1667, A 0.000, B 0.000, C 0.000 }
gfCNCPoint1[24333] = {X 209.4842, Y 61.4084, Z -2.1667, A 0.000, B 0.000, C 0.000 }
gfCNCPoint1[24334] = {X 209.1644, Y 60.2149, Z -2.1667, A 0.000, B 0.000, C 0.000 }
gfCNCPoint1[24335] = {X 209.0510, Y 58.9845, Z -2.1667, A 0.000, B 0.000, C 0.000 }
gfCNCPoint1[24336] = {X 209.0508, Y 58.0000, Z -2.1667, A 0.000, B 0.000, C 0.000 }
gfCNCPoint1[24337] = {X 209.1477, Y 56.8162, Z -2.1667, A 0.000, B 0.000, C 0.000 }
gfCNCPoint1[24338] = {X 209.4358, Y 55.6638, Z -2.1667, A 0.000, B 0.000, C 0.000 }
gfCNCPoint1[24339] = {X 209.9075, Y 54.5737, Z -2.1667, A 0.000, B 0.000, C 0.000 }
gfCNCPoint1[24340] = {X 210.5502, Y 53.5748, Z -2.1667, A 0.000, B 0.000, C 0.000 }
gfCNCPoint1[24341] = {X 211.3467, Y 52.6937, Z -2.1667, A 0.000, B 0.000, C 0.000 }
gfCNCPoint1[24342] = {X 212.2759, Y 51.9538, Z -2.1667, A 0.000, B 0.000, C 0.000 }
gfCNCPoint1[24343] = {X 213.3131, Y 51.3749, Z -2.1667, A 0.000, B 0.000, C 0.000 }
gfCNCPoint1[24344] = {X 214.4306, Y 50.9724, Z -2.1667, A 0.000, B 0.000, C 0.000 }
gfCNCPoint1[24345] = {X 215.3724, Y 50.7834, Z -2.1667, A 0.000, B 0.000, C 0.000 }
gfCNCPoint1[24346] = {X 216.3308, Y 50.7200, Z -2.1667, A 0.000, B 0.000, C 0.000 }
gfCNCPoint1[24347] = {X 237.2617, Y 50.7200, Z -2.1667, A 0.000, B 0.000, C 0.000 }
gfCNCPoint1[24348] = {X 238.3057, Y 50.7953, Z -2.1667, A 0.000, B 0.000, C 0.000 }
gfCNCPoint1[24349] = {X 239.3282, Y 51.0195, Z -2.1667, A 0.000, B 0.000, C 0.000 }
gfCNCPoint1[24350] = {X 240.3080, Y 51.3880, Z -2.1667, A 0.000, B 0.000, C 0.000 }
gfCNCPoint1[24351] = {X 241.2247, Y 51.8932, Z -2.1667, A 0.000, B 0.000, C 0.000 }
gfCNCPoint1[24352] = {X 242.0742, Y 52.5376, Z -2.1667, A 0.000, B 0.000, C 0.000 }
gfCNCPoint1[24353] = {X 242.8204, Y 53.2991, Z -2.1667, A 0.000, B 0.000, C 0.000 }
gfCNCPoint1[24354] = {X 243.4474, Y 54.1614, Z -2.1667, A 0.000, B 0.000, C 0.000 }
gfCNCPoint1[24355] = {X 243.9418, Y 55.1061, Z -2.1667, A 0.000, B 0.000, C 0.000 }
gfCNCPoint1[24356] = {X 244.2928, Y 56.1128, Z -2.1667, A 0.000, B 0.000, C 0.000 }
gfCNCPoint1[24357] = {X 248.5776, Y 57.7833, Z -2.1667, A 0.000, B 0.000, C 0.000 }
gfCNCPoint1[24358] = {X 272.6734, Y 67.3439, Z -2.1667, A 0.000, B 0.000, C 0.000 }
gfCNCPoint1[24359] = {X 272.6732, Y 65.2845, Z -2.1667, A 0.000, B 0.000, C 0.000 }
gfCNCPoint1[24360] = {X 271.6658, Y 64.6035, Z -2.1667, A 0.000, B 0.000, C 0.000 }
gfCNCPoint1[24361] = {X 270.7858, Y 63.7642, Z -2.1667, A 0.000, B 0.000, C 0.000 }
gfCNCPoint1[24362] = {X 270.0578, Y 62.7902, Z -2.1667, A 0.000, B 0.000, C 0.000 }
gfCNCPoint1[24363] = {X 269.5021, Y 61.7085, Z -2.1667, A 0.000, B 0.000, C 0.000 }
gfCNCPoint1[24364] = {X 269.2030, Y 60.8265, Z -2.1667, A 0.000, B 0.000, C 0.000 }
gfCNCPoint1[24365] = {X 269.0189, Y 59.9135, Z -2.1667, A 0.000, B 0.000, C 0.000 }
gfCNCPoint1[24366] = {X 268.9529, Y 58.9845, Z -2.1667, A 0.000, B 0.000, C 0.000 }
gfCNCPoint1[24367] = {X 268.9527, Y 58.0000, Z -2.1667, A 0.000, B 0.000, C 0.000 }
gfCNCPoint1[24368] = {X 269.0633, Y 56.7358, Z -2.1667, A 0.000, B 0.000, C 0.000 }
gfCNCPoint1[24369] = {X 269.3917, Y 55.5101, Z -2.1667, A 0.000, B 0.000, C 0.000 }
gfCNCPoint1[24370] = {X 269.9280, Y 54.3600, Z -2.1667, A 0.000, B 0.000, C 0.000 }
gfCNCPoint1[24371] = {X 270.6559, Y 53.3205, Z -2.1667, A 0.000, B 0.000, C 0.000 }
gfCNCPoint1[24372] = {X 271.5532, Y 52.4232, Z -2.1667, A 0.000, B 0.000, C 0.000 }
gfCNCPoint1[24373] = {X 272.5927, Y 51.6953, Z -2.1667, A 0.000, B 0.000, C 0.000 }
gfCNCPoint1[24374] = {X 273.7428, Y 51.1590, Z -2.1667, A 0.000, B 0.000, C 0.000 }
gfCNCPoint1[24375] = {X 274.9685, Y 50.8306, Z -2.1667, A 0.000, B 0.000, C 0.000 }
gfCNCPoint1[24376] = {X 276.2327, Y 50.7200, Z -2.1667, A 0.000, B 0.000, C 0.000 }
gfCNCPoint1[24377] = {X 292.7731, Y 50.7200, Z -2.1667, A 0.000, B 0.000, C 0.000 }
gfCNCPoint1[24378] = {X 293.4209, Y 50.7489, Z -2.1667, A 0.000, B 0.000, C 0.000 }
gfCNCPoint1[24379] = {X 294.0636, Y 50.8353, Z -2.1667, A 0.000, B 0.000, C 0.000 }
gfCNCPoint1[24380] = {X 294.7296, Y 50.9878, Z -2.1667, A 0.000, B 0.000, C 0.000 }
gfCNCPoint1[24381] = {X 295.3783, Y 51.2021, Z -2.1667, A 0.000, B 0.000, C 0.000 }
gfCNCPoint1[24382] = {X 298.3089, Y 43.5556, Z -2.1667, A 0.000, B 0.000, C 0.000 }
gfCNCPoint1[24383] = {X 298.4822, Y 42.5316, Z -2.1667, A 0.000, B 0.000, C 0.000 }
gfCNCPoint1[24384] = {X 298.7929, Y 41.5406, Z -2.1667, A 0.000, B 0.000, C 0.000 }
gfCNCPoint1[24385] = {X 299.2351, Y 40.6008, Z -2.1667, A 0.000, B 0.000, C 0.000 }
gfCNCPoint1[24386] = {X 299.8007, Y 39.7298, Z -2.1667, A 0.000, B 0.000, C 0.000 }
gfCNCPoint1[24387] = {X 299.8007, Y 36.9943, Z -2.1667, A 0.000, B 0.000, C 0.000 }
gfCNCPoint1[24388] = {X 296.8133, Y 36.9943, Z -2.1667, A 0.000, B 0.000, C 0.000 }
gfCNCPoint1[24389] = {X 296.8129, Y 39.7491, Z -2.1667, A 0.000, B 0.000, C 0.000 }
gfCNCPoint1[24390] = {X 297.3845, Y 40.6121, Z -2.1667, A 0.000, B 0.000, C 0.000 }
gfCNCPoint1[24391] = {X 297.8298, Y 41.5467, Z -2.1667, A 0.000, B 0.000, C 0.000 }
gfCNCPoint1[24392] = {X 298.1399, Y 42.5343, Z -2.1667, A 0.000, B 0.000, C 0.000 }
gfCNCPoint1[24393] = {X 298.3089, Y 43.5556, Z -2.1667, A 0.000, B 0.000, C 0.000 }
gfCNCPoint1[24394] = {X 296.2372, Y 48.9611, Z -2.1667, A 0.000, B 0.000, C 0.000 }
gfCNCPoint1[24395] = {X 296.6128, Y 49.1141, Z -2.1667, A 0.000, B 0.000, C 0.000 }
gfCNCPoint1[24396] = {X 296.9817, Y 49.2828, Z -2.1667, A 0.000, B 0.000, C 0.000 }
gfCNCPoint1[24397] = {X 297.2571, Y 49.4212, Z -2.1667, A 0.000, B 0.000, C 0.000 }
gfCNCPoint1[24398] = {X 297.5280, Y 49.5683, Z -2.1667, A 0.000, B 0.000, C 0.000 }
gfCNCPoint1[24399] = {X 298.7174, Y 50.3602, Z -2.1667, A 0.000, B 0.000, C 0.000 }
gfCNCPoint1[24400] = {X 299.7774, Y 51.3185, Z -2.1667, A 0.000, B 0.000, C 0.000 }
gfCNCPoint1[24401] = {X 300.6847, Y 52.4224, Z -2.1667, A 0.000, B 0.000, C 0.000 }
gfCNCPoint1[24402] = {X 301.5914, Y 51.3191, Z -2.1667, A 0.000, B 0.000, C 0.000 }
gfCNCPoint1[24403] = {X 302.6506, Y 50.3611, Z -2.1667, A 0.000, B 0.000, C 0.000 }
gfCNCPoint1[24404] = {X 303.8393, Y 49.5695, Z -2.1667, A 0.000, B 0.000, C 0.000 }
gfCNCPoint1[24405] = {X 302.8989, Y 49.0956, Z -2.1667, A 0.000, B 0.000, C 0.000 }
gfCNCPoint1[24406] = {X 302.0820, Y 48.4310, Z -2.1667, A 0.000, B 0.000, C 0.000 }
gfCNCPoint1[24407] = {X 301.4268, Y 47.6067, Z -2.1667, A 0.000, B 0.000, C 0.000 }
gfCNCPoint1[24408] = {X 300.9636, Y 46.6610, Z -2.1667, A 0.000, B 0.000, C 0.000 }
gfCNCPoint1[24409] = {X 300.7923, Y 46.0759, Z -2.1667, A 0.000, B 0.000, C 0.000 }
gfCNCPoint1[24410] = {X 300.6953, Y 45.4741, Z -2.1667, A 0.000, B 0.000, C 0.000 }
gfCNCPoint1[24411] = {X 300.6790, Y 45.2570, Z -2.1667, A 0.000, B 0.000, C 0.000 }
gfCNCPoint1[24412] = {X 300.6724, Y 45.0393, Z -2.1667, A 0.000, B 0.000, C 0.000 }
gfCNCPoint1[24413] = {X 300.6725, Y 44.1874, Z -2.1667, A 0.000, B 0.000, C 0.000 }
gfCNCPoint1[24414] = {X 300.6810, Y 43.9907, Z -2.1667, A 0.000, B 0.000, C 0.000 }
gfCNCPoint1[24415] = {X 300.6969, Y 43.7944, Z -2.1667, A 0.000, B 0.000, C 0.000 }
gfCNCPoint1[24416] = {X 300.8618, Y 42.9144, Z -2.1667, A 0.000, B 0.000, C 0.000 }
gfCNCPoint1[24417] = {X 301.1742, Y 42.0753, Z -2.1667, A 0.000, B 0.000, C 0.000 }
gfCNCPoint1[24418] = {X 301.6249, Y 41.3017, Z -2.1667, A 0.000, B 0.000, C 0.000 }
gfCNCPoint1[24419] = {X 302.2007, Y 40.6161, Z -2.1667, A 0.000, B 0.000, C 0.000 }
gfCNCPoint1[24420] = {X 302.2007, Y 34.5943, Z -2.1667, A 0.000, B 0.000, C 0.000 }
gfCNCPoint1[24421] = {X 294.4137, Y 34.5943, Z -2.1667, A 0.000, B 0.000, C 0.000 }
gfCNCPoint1[24422] = {X 294.4128, Y 40.6559, Z -2.1667, A 0.000, B 0.000, C 0.000 }
gfCNCPoint1[24423] = {X 294.9934, Y 41.3233, Z -2.1667, A 0.000, B 0.000, C 0.000 }
gfCNCPoint1[24424] = {X 295.4468, Y 42.0828, Z -2.1667, A 0.000, B 0.000, C 0.000 }
gfCNCPoint1[24425] = {X 295.7587, Y 42.9105, Z -2.1667, A 0.000, B 0.000, C 0.000 }
gfCNCPoint1[24426] = {X 295.9194, Y 43.7803, Z -2.1667, A 0.000, B 0.000, C 0.000 }
gfCNCPoint1[24427] = {X 295.9349, Y 43.9944, Z -2.1667, A 0.000, B 0.000, C 0.000 }
gfCNCPoint1[24428] = {X 295.9411, Y 44.2089, Z -2.1667, A 0.000, B 0.000, C 0.000 }
gfCNCPoint1[24429] = {X 295.9411, Y 45.0000, Z -2.1667, A 0.000, B 0.000, C 0.000 }
gfCNCPoint1[24430] = {X 295.9354, Y 45.2373, Z -2.1667, A 0.000, B 0.000, C 0.000 }
gfCNCPoint1[24431] = {X 295.9180, Y 45.4741, Z -2.1667, A 0.000, B 0.000, C 0.000 }
gfCNCPoint1[24432] = {X 298.3067, Y 45.7073, Z -2.1667, A 0.000, B 0.000, C 0.000 }
gfCNCPoint1[24433] = {X 298.2010, Y 46.4214, Z -2.1667, A 0.000, B 0.000, C 0.000 }
gfCNCPoint1[24434] = {X 298.0252, Y 47.1215, Z -2.1667, A 0.000, B 0.000, C 0.000 }
gfCNCPoint1[24435] = {X 298.3689, Y 47.2942, Z -2.1667, A 0.000, B 0.000, C 0.000 }
gfCNCPoint1[24436] = {X 298.7069, Y 47.4778, Z -2.1667, A 0.000, B 0.000, C 0.000 }
gfCNCPoint1[24437] = {X 298.4514, Y 46.6051, Z -2.1667, A 0.000, B 0.000, C 0.000 }
gfCNCPoint1[24438] = {X 298.3067, Y 45.7073, Z -2.1667, A 0.000, B 0.000, C 0.000 }
gfCNCPoint1[24439] = {X 295.9180, Y 45.4741, Z -2.1667, A 0.000, B 0.000, C 0.000 }
gfCNCPoint1[24440] = {X 295.8472, Y 45.9528, Z -2.1667, A 0.000, B 0.000, C 0.000 }
gfCNCPoint1[24441] = {X 295.7293, Y 46.4221, Z -2.1667, A 0.000, B 0.000, C 0.000 }
gfCNCPoint1[24442] = {X 295.4314, Y 47.1714, Z -2.1667, A 0.000, B 0.000, C 0.000 }
gfCNCPoint1[24443] = {X 295.0142, Y 47.8614, Z -2.1667, A 0.000, B 0.000, C 0.000 }
gfCNCPoint1[24444] = {X 294.4890, Y 48.4733, Z -2.1667, A 0.000, B 0.000, C 0.000 }
gfCNCPoint1[24445] = {X 295.3746, Y 48.6761, Z -2.1667, A 0.000, B 0.000, C 0.000 }
gfCNCPoint1[24446] = {X 296.2372, Y 48.9611, Z -2.1667, A 0.000, B 0.000, C 0.000 }
gfCNCPoint1[24447] = {X 295.3783, Y 51.2021, Z -2.1667, A 0.000, B 0.000, C 0.000 }
gfCNCPoint1[24448] = {X 296.3503, Y 51.6595, Z -2.1667, A 0.000, B 0.000, C 0.000 }
gfCNCPoint1[24449] = {X 297.2444, Y 52.2549, Z -2.1667, A 0.000, B 0.000, C 0.000 }
gfCNCPoint1[24450] = {X 298.0411, Y 52.9754, Z -2.1667, A 0.000, B 0.000, C 0.000 }
gfCNCPoint1[24451] = {X 298.7231, Y 53.8053, Z -2.1667, A 0.000, B 0.000, C 0.000 }
gfCNCPoint1[24452] = {X 299.2946, Y 54.7645, Z -2.1667, A 0.000, B 0.000, C 0.000 }
gfCNCPoint1[24453] = {X 299.7126, Y 55.7997, Z -2.1667, A 0.000, B 0.000, C 0.000 }
gfCNCPoint1[24454] = {X 299.9675, Y 56.8868, Z -2.1667, A 0.000, B 0.000, C 0.000 }
gfCNCPoint1[24455] = {X 300.0531, Y 58.0000, Z -2.1667, A 0.000, B 0.000, C 0.000 }
gfCNCPoint1[24456] = {X 300.0531, Y 58.9455, Z -2.1667, A 0.000, B 0.000, C 0.000 }
gfCNCPoint1[24457] = {X 299.9644, Y 60.0548, Z -2.1667, A 0.000, B 0.000, C 0.000 }
gfCNCPoint1[24458] = {X 299.7080, Y 61.1376, Z -2.1667, A 0.000, B 0.000, C 0.000 }
gfCNCPoint1[24459] = {X 299.2900, Y 62.1689, Z -2.1667, A 0.000, B 0.000, C 0.000 }
gfCNCPoint1[24460] = {X 298.7201, Y 63.1246, Z -2.1667, A 0.000, B 0.000, C 0.000 }
gfCNCPoint1[24461] = {X 300.6817, Y 64.5074, Z -2.1667, A 0.000, B 0.000, C 0.000 }
gfCNCPoint1[24462] = {X 299.7819, Y 65.6038, Z -2.1667, A 0.000, B 0.000, C 0.000 }
gfCNCPoint1[24463] = {X 298.7318, Y 66.5571, Z -2.1667, A 0.000, B 0.000, C 0.000 }
gfCNCPoint1[24464] = {X 298.7318, Y 89.4424, Z -2.1667, A 0.000, B 0.000, C 0.000 }
gfCNCPoint1[24465] = {X 299.8285, Y 90.4467, Z -2.1667, A 0.000, B 0.000, C 0.000 }
gfCNCPoint1[24466] = {X 300.7592, Y 91.6066, Z -2.1667, A 0.000, B 0.000, C 0.000 }
gfCNCPoint1[24467] = {X 301.5018, Y 92.8949, Z -2.1667, A 0.000, B 0.000, C 0.000 }
gfCNCPoint1[24468] = {X 304.0678, Y 92.8949, Z -2.1667, A 0.000, B 0.000, C 0.000 }
gfCNCPoint1[24469] = {X 303.7101, Y 91.8992, Z -2.1667, A 0.000, B 0.000, C 0.000 }
gfCNCPoint1[24470] = {X 303.4141, Y 90.8834, Z -2.1667, A 0.000, B 0.000, C 0.000 }
gfCNCPoint1[24471] = {X 302.9751, Y 88.8125, Z -2.1667, A 0.000, B 0.000, C 0.000 }
gfCNCPoint1[24472] = {X 302.7153, Y 86.7116, Z -2.1667, A 0.000, B 0.000, C 0.000 }
gfCNCPoint1[24473] = {X 302.6364, Y 84.5962, Z -2.1667, A 0.000, B 0.000, C 0.000 }
gfCNCPoint1[24474] = {X 302.6376, Y 83.2276, Z -2.1667, A 0.000, B 0.000, C 0.000 }
gfCNCPoint1[24475] = {X 302.6376, Y 66.5628, Z -2.1667, A 0.000, B 0.000, C 0.000 }
gfCNCPoint1[24476] = {X 301.5839, Y 65.6072, Z -2.1667, A 0.000, B 0.000, C 0.000 }
gfCNCPoint1[24477] = {X 300.6817, Y 64.5074, Z -2.1667, A 0.000, B 0.000, C 0.000 }
gfCNCPoint1[24478] = {X 298.7201, Y 63.1246, Z -2.1667, A 0.000, B 0.000, C 0.000 }
gfCNCPoint1[24479] = {X 298.0339, Y 63.9592, Z -2.1667, A 0.000, B 0.000, C 0.000 }
gfCNCPoint1[24480] = {X 297.2319, Y 64.6833, Z -2.1667, A 0.000, B 0.000, C 0.000 }
gfCNCPoint1[24481] = {X 296.3318, Y 65.2810, Z -2.1667, A 0.000, B 0.000, C 0.000 }
gfCNCPoint1[24482] = {X 296.3318, Y 90.7169, Z -2.1667, A 0.000, B 0.000, C 0.000 }
gfCNCPoint1[24483] = {X 297.3120, Y 91.3795, Z -2.1667, A 0.000, B 0.000, C 0.000 }
gfCNCPoint1[24484] = {X 298.1726, Y 92.1914, Z -2.1667, A 0.000, B 0.000, C 0.000 }
gfCNCPoint1[24485] = {X 298.8909, Y 93.1315, Z -2.1667, A 0.000, B 0.000, C 0.000 }
gfCNCPoint1[24486] = {X 299.4483, Y 94.1751, Z -2.1667, A 0.000, B 0.000, C 0.000 }
gfCNCPoint1[24487] = {X 299.8301, Y 95.2949, Z -2.1667, A 0.000, B 0.000, C 0.000 }
gfCNCPoint1[24488] = {X 308.0995, Y 95.2949, Z -2.1667, A 0.000, B 0.000, C 0.000 }
gfCNCPoint1[24489] = {X 307.0964, Y 93.7117, Z -2.1667, A 0.000, B 0.000, C 0.000 }
gfCNCPoint1[24490] = {X 306.3006, Y 92.0148, Z -2.1667, A 0.000, B 0.000, C 0.000 }
gfCNCPoint1[24491] = {X 305.9926, Y 91.1575, Z -2.1667, A 0.000, B 0.000, C 0.000 }
gfCNCPoint1[24492] = {X 305.7378, Y 90.2829, Z -2.1667, A 0.000, B 0.000, C 0.000 }
gfCNCPoint1[24493] = {X 305.3416, Y 88.4124, Z -2.1667, A 0.000, B 0.000, C 0.000 }
gfCNCPoint1[24494] = {X 305.1072, Y 86.5149, Z -2.1667, A 0.000, B 0.000, C 0.000 }
gfCNCPoint1[24495] = {X 305.0364, Y 84.6042, Z -2.1667, A 0.000, B 0.000, C 0.000 }
gfCNCPoint1[24496] = {X 305.0376, Y 83.2289, Z -2.1667, A 0.000, B 0.000, C 0.000 }
gfCNCPoint1[24497] = {X 305.0376, Y 65.2850, Z -2.1667, A 0.000, B 0.000, C 0.000 }
gfCNCPoint1[24498] = {X 304.1352, Y 64.6871, Z -2.1667, A 0.000, B 0.000, C 0.000 }
gfCNCPoint1[24499] = {X 303.3314, Y 63.9619, Z -2.1667, A 0.000, B 0.000, C 0.000 }
gfCNCPoint1[24500] = {X 302.6440, Y 63.1256, Z -2.1667, A 0.000, B 0.000, C 0.000 }
gfCNCPoint1[24501] = {X 302.0790, Y 62.1783, Z -2.1667, A 0.000, B 0.000, C 0.000 }
gfCNCPoint1[24502] = {X 301.6637, Y 61.1565, Z -2.1667, A 0.000, B 0.000, C 0.000 }
gfCNCPoint1[24503] = {X 301.4076, Y 60.0837, Z -2.1667, A 0.000, B 0.000, C 0.000 }
gfCNCPoint1[24504] = {X 301.3164, Y 58.9845, Z -2.1667, A 0.000, B 0.000, C 0.000 }
gfCNCPoint1[24505] = {X 301.3162, Y 58.0000, Z -2.1667, A 0.000, B 0.000, C 0.000 }
gfCNCPoint1[24506] = {X 301.4018, Y 56.8868, Z -2.1667, A 0.000, B 0.000, C 0.000 }
gfCNCPoint1[24507] = {X 301.6567, Y 55.7997, Z -2.1667, A 0.000, B 0.000, C 0.000 }
gfCNCPoint1[24508] = {X 302.0747, Y 54.7645, Z -2.1667, A 0.000, B 0.000, C 0.000 }
gfCNCPoint1[24509] = {X 302.6462, Y 53.8053, Z -2.1667, A 0.000, B 0.000, C 0.000 }
gfCNCPoint1[24510] = {X 303.3281, Y 52.9755, Z -2.1667, A 0.000, B 0.000, C 0.000 }
gfCNCPoint1[24511] = {X 304.1247, Y 52.2551, Z -2.1667, A 0.000, B 0.000, C 0.000 }
gfCNCPoint1[24512] = {X 305.0187, Y 51.6597, Z -2.1667, A 0.000, B 0.000, C 0.000 }
gfCNCPoint1[24513] = {X 306.1514, Y 51.1428, Z -2.1667, A 0.000, B 0.000, C 0.000 }
gfCNCPoint1[24514] = {X 307.3557, Y 50.8265, Z -2.1667, A 0.000, B 0.000, C 0.000 }
gfCNCPoint1[24515] = {X 308.5962, Y 50.7200, Z -2.1667, A 0.000, B 0.000, C 0.000 }
gfCNCPoint1[24516] = {X 324.3107, Y 50.7200, Z -2.1667, A 0.000, B 0.000, C 0.000 }
gfCNCPoint1[24517] = {X 325.2469, Y 50.7804, Z -2.1667, A 0.000, B 0.000, C 0.000 }
gfCNCPoint1[24518] = {X 326.1675, Y 50.9608, Z -2.1667, A 0.000, B 0.000, C 0.000 }
gfCNCPoint1[24519] = {X 326.5260, Y 51.0653, Z -2.1667, A 0.000, B 0.000, C 0.000 }
gfCNCPoint1[24520] = {X 326.8787, Y 51.1880, Z -2.1667, A 0.000, B 0.000, C 0.000 }
gfCNCPoint1[24521] = {X 327.4571, Y 51.4350, Z -2.1667, A 0.000, B 0.000, C 0.000 }
gfCNCPoint1[24522] = {X 328.0120, Y 51.7311, Z -2.1667, A 0.000, B 0.000, C 0.000 }
gfCNCPoint1[24523] = {X 328.5424, Y 52.0762, Z -2.1667, A 0.000, B 0.000, C 0.000 }
gfCNCPoint1[24524] = {X 329.0409, Y 52.4661, Z -2.1667, A 0.000, B 0.000, C 0.000 }
gfCNCPoint1[24525] = {X 329.9215, Y 53.3614, Z -2.1667, A 0.000, B 0.000, C 0.000 }
gfCNCPoint1[24526] = {X 330.6352, Y 54.3946, Z -2.1667, A 0.000, B 0.000, C 0.000 }
gfCNCPoint1[24527] = {X 331.1607, Y 55.5351, Z -2.1667, A 0.000, B 0.000, C 0.000 }
gfCNCPoint1[24528] = {X 331.4824, Y 56.7489, Z -2.1667, A 0.000, B 0.000, C 0.000 }
gfCNCPoint1[24529] = {X 331.5907, Y 58.0000, Z -2.1667, A 0.000, B 0.000, C 0.000 }
gfCNCPoint1[24530] = {X 331.5907, Y 58.9402, Z -2.1667, A 0.000, B 0.000, C 0.000 }
gfCNCPoint1[24531] = {X 331.4730, Y 60.2170, Z -2.1667, A 0.000, B 0.000, C 0.000 }
gfCNCPoint1[24532] = {X 331.1343, Y 61.4537, Z -2.1667, A 0.000, B 0.000, C 0.000 }
gfCNCPoint1[24533] = {X 330.5850, Y 62.6123, Z -2.1667, A 0.000, B 0.000, C 0.000 }
gfCNCPoint1[24534] = {X 329.8419, Y 63.6572, Z -2.1667, A 0.000, B 0.000, C 0.000 }
gfCNCPoint1[24535] = {X 328.9279, Y 64.5565, Z -2.1667, A 0.000, B 0.000, C 0.000 }
gfCNCPoint1[24536] = {X 327.8710, Y 65.2825, Z -2.1667, A 0.000, B 0.000, C 0.000 }
gfCNCPoint1[24537] = {X 327.8722, Y 83.2150, Z -2.1667, A 0.000, B 0.000, C 0.000 }
gfCNCPoint1[24538] = {X 327.8857, Y 84.5924, Z -2.1667, A 0.000, B 0.000, C 0.000 }
gfCNCPoint1[24539] = {X 327.8950, Y 84.9547, Z -2.1667, A 0.000, B 0.000, C 0.000 }
gfCNCPoint1[24540] = {X 327.9219, Y 85.3161, Z -2.1667, A 0.000, B 0.000, C 0.000 }
gfCNCPoint1[24541] = {X 328.8634, Y 85.6738, Z -2.1667, A 0.000, B 0.000, C 0.000 }
gfCNCPoint1[24542] = {X 329.8332, Y 85.9453, Z -2.1667, A 0.000, B 0.000, C 0.000 }
gfCNCPoint1[24543] = {X 332.7043, Y 86.5207, Z -2.1667, A 0.000, B 0.000, C 0.000 }
gfCNCPoint1[24544] = {X 335.6093, Y 86.8871, Z -2.1667, A 0.000, B 0.000, C 0.000 }
gfCNCPoint1[24545] = {X 339.6588, Y 87.1997, Z -2.1667, A 0.000, B 0.000, C 0.000 }
gfCNCPoint1[24546] = {X 343.7164, Y 87.3755, Z -2.1667, A 0.000, B 0.000, C 0.000 }
gfCNCPoint1[24547] = {X 347.7777, Y 87.4143, Z -2.1667, A 0.000, B 0.000, C 0.000 }
gfCNCPoint1[24548] = {X 352.0650, Y 87.3776, Z -2.1667, A 0.000, B 0.000, C 0.000 }
gfCNCPoint1[24549] = {X 356.3481, Y 87.1863, Z -2.1667, A 0.000, B 0.000, C 0.000 }
gfCNCPoint1[24550] = {X 360.6216, Y 86.8408, Z -2.1667, A 0.000, B 0.000, C 0.000 }
gfCNCPoint1[24551] = {X 362.7646, Y 86.5747, Z -2.1667, A 0.000, B 0.000, C 0.000 }
gfCNCPoint1[24552] = {X 364.8876, Y 86.1799, Z -2.1667, A 0.000, B 0.000, C 0.000 }
gfCNCPoint1[24553] = {X 366.9831, Y 85.6579, Z -2.1667, A 0.000, B 0.000, C 0.000 }
gfCNCPoint1[24554] = {X 367.4433, Y 85.5114, Z -2.1667, A 0.000, B 0.000, C 0.000 }
gfCNCPoint1[24555] = {X 367.8898, Y 85.3271, Z -2.1667, A 0.000, B 0.000, C 0.000 }
gfCNCPoint1[24556] = {X 367.9433, Y 84.5784, Z -2.1667, A 0.000, B 0.000, C 0.000 }
gfCNCPoint1[24557] = {X 367.9611, Y 83.8280, Z -2.1667, A 0.000, B 0.000, C 0.000 }
gfCNCPoint1[24558] = {X 367.9596, Y 65.2844, Z -2.1667, A 0.000, B 0.000, C 0.000 }
gfCNCPoint1[24559] = {X 366.9055, Y 64.5654, Z -2.1667, A 0.000, B 0.000, C 0.000 }
gfCNCPoint1[24560] = {X 365.9932, Y 63.6733, Z -2.1667, A 0.000, B 0.000, C 0.000 }
gfCNCPoint1[24561] = {X 365.2506, Y 62.6357, Z -2.1667, A 0.000, B 0.000, C 0.000 }
gfCNCPoint1[24562] = {X 364.7006, Y 61.4844, Z -2.1667, A 0.000, B 0.000, C 0.000 }
gfCNCPoint1[24563] = {X 364.3601, Y 60.2547, Z -2.1667, A 0.000, B 0.000, C 0.000 }
gfCNCPoint1[24564] = {X 364.2395, Y 58.9845, Z -2.1667, A 0.000, B 0.000, C 0.000 }
gfCNCPoint1[24565] = {X 364.2393, Y 58.0000, Z -2.1667, A 0.000, B 0.000, C 0.000 }
gfCNCPoint1[24566] = {X 364.3499, Y 56.7358, Z -2.1667, A 0.000, B 0.000, C 0.000 }
gfCNCPoint1[24567] = {X 364.6783, Y 55.5101, Z -2.1667, A 0.000, B 0.000, C 0.000 }
gfCNCPoint1[24568] = {X 365.2146, Y 54.3600, Z -2.1667, A 0.000, B 0.000, C 0.000 }
gfCNCPoint1[24569] = {X 365.9425, Y 53.3205, Z -2.1667, A 0.000, B 0.000, C 0.000 }
gfCNCPoint1[24570] = {X 366.8398, Y 52.4232, Z -2.1667, A 0.000, B 0.000, C 0.000 }
gfCNCPoint1[24571] = {X 367.8793, Y 51.6953, Z -2.1667, A 0.000, B 0.000, C 0.000 }
gfCNCPoint1[24572] = {X 369.0294, Y 51.1590, Z -2.1667, A 0.000, B 0.000, C 0.000 }
gfCNCPoint1[24573] = {X 370.2551, Y 50.8306, Z -2.1667, A 0.000, B 0.000, C 0.000 }
gfCNCPoint1[24574] = {X 371.5193, Y 50.7200, Z -2.1667, A 0.000, B 0.000, C 0.000 }
gfCNCPoint1[24575] = {X 388.0597, Y 50.7200, Z -2.1667, A 0.000, B 0.000, C 0.000 }
gfCNCPoint1[24576] = {X 389.2271, Y 50.8142, Z -2.1667, A 0.000, B 0.000, C 0.000 }
gfCNCPoint1[24577] = {X 390.3643, Y 51.0944, Z -2.1667, A 0.000, B 0.000, C 0.000 }
gfCNCPoint1[24578] = {X 391.4418, Y 51.5533, Z -2.1667, A 0.000, B 0.000, C 0.000 }
gfCNCPoint1[24579] = {X 392.4319, Y 52.1791, Z -2.1667, A 0.000, B 0.000, C 0.000 }
gfCNCPoint1[24580] = {X 393.3087, Y 52.9556, Z -2.1667, A 0.000, B 0.000, C 0.000 }
gfCNCPoint1[24581] = {X 394.1855, Y 52.1791, Z -2.1667, A 0.000, B 0.000, C 0.000 }
gfCNCPoint1[24582] = {X 395.1756, Y 51.5533, Z -2.1667, A 0.000, B 0.000, C 0.000 }
gfCNCPoint1[24583] = {X 396.2531, Y 51.0944, Z -2.1667, A 0.000, B 0.000, C 0.000 }
gfCNCPoint1[24584] = {X 397.3903, Y 50.8142, Z -2.1667, A 0.000, B 0.000, C 0.000 }
gfCNCPoint1[24585] = {X 398.5577, Y 50.7200, Z -2.1667, A 0.000, B 0.000, C 0.000 }
gfCNCPoint1[24586] = {X 419.4886, Y 50.7200, Z -2.1667, A 0.000, B 0.000, C 0.000 }
gfCNCPoint1[24587] = {X 420.6741, Y 50.8172, Z -2.1667, A 0.000, B 0.000, C 0.000 }
gfCNCPoint1[24588] = {X 421.8279, Y 51.1061, Z -2.1667, A 0.000, B 0.000, C 0.000 }
gfCNCPoint1[24589] = {X 422.9192, Y 51.5790, Z -2.1667, A 0.000, B 0.000, C 0.000 }
gfCNCPoint1[24590] = {X 423.9190, Y 52.2233, Z -2.1667, A 0.000, B 0.000, C 0.000 }
gfCNCPoint1[24591] = {X 424.8005, Y 53.0219, Z -2.1667, A 0.000, B 0.000, C 0.000 }
gfCNCPoint1[24592] = {X 425.5403, Y 53.9533, Z -2.1667, A 0.000, B 0.000, C 0.000 }
gfCNCPoint1[24593] = {X 426.1184, Y 54.9927, Z -2.1667, A 0.000, B 0.000, C 0.000 }
gfCNCPoint1[24594] = {X 426.5196, Y 56.1125, Z -2.1667, A 0.000, B 0.000, C 0.000 }
gfCNCPoint1[24595] = {X 430.7007, Y 57.7420, Z -2.1667, A 0.000, B 0.000, C 0.000 }
gfCNCPoint1[24596] = {X 454.9004, Y 67.3431, Z -2.1667, A 0.000, B 0.000, C 0.000 }
gfCNCPoint1[24597] = {X 454.9001, Y 65.2845, Z -2.1667, A 0.000, B 0.000, C 0.000 }
gfCNCPoint1[24598] = {X 453.8926, Y 64.6034, Z -2.1667, A 0.000, B 0.000, C 0.000 }
gfCNCPoint1[24599] = {X 453.0125, Y 63.7640, Z -2.1667, A 0.000, B 0.000, C 0.000 }
gfCNCPoint1[24600] = {X 452.2845, Y 62.7898, Z -2.1667, A 0.000, B 0.000, C 0.000 }
gfCNCPoint1[24601] = {X 451.7288, Y 61.7080, Z -2.1667, A 0.000, B 0.000, C 0.000 }
gfCNCPoint1[24602] = {X 451.4298, Y 60.8261, Z -2.1667, A 0.000, B 0.000, C 0.000 }
gfCNCPoint1[24603] = {X 451.2458, Y 59.9133, Z -2.1667, A 0.000, B 0.000, C 0.000 }
gfCNCPoint1[24604] = {X 451.1798, Y 58.9845, Z -2.1667, A 0.000, B 0.000, C 0.000 }
gfCNCPoint1[24605] = {X 451.1796, Y 58.0000, Z -2.1667, A 0.000, B 0.000, C 0.000 }
gfCNCPoint1[24606] = {X 451.2795, Y 56.7981, Z -2.1667, A 0.000, B 0.000, C 0.000 }
gfCNCPoint1[24607] = {X 451.5765, Y 55.6291, Z -2.1667, A 0.000, B 0.000, C 0.000 }
gfCNCPoint1[24608] = {X 452.0624, Y 54.5253, Z -2.1667, A 0.000, B 0.000, C 0.000 }
gfCNCPoint1[24609] = {X 452.7238, Y 53.5168, Z -2.1667, A 0.000, B 0.000, C 0.000 }
gfCNCPoint1[24610] = {X 453.5427, Y 52.6313, Z -2.1667, A 0.000, B 0.000, C 0.000 }
gfCNCPoint1[24611] = {X 454.4966, Y 51.8932, Z -2.1667, A 0.000, B 0.000, C 0.000 }
gfCNCPoint1[24612] = {X 455.4133, Y 51.3880, Z -2.1667, A 0.000, B 0.000, C 0.000 }
gfCNCPoint1[24613] = {X 456.3931, Y 51.0195, Z -2.1667, A 0.000, B 0.000, C 0.000 }
gfCNCPoint1[24614] = {X 457.4155, Y 50.7953, Z -2.1667, A 0.000, B 0.000, C 0.000 }
gfCNCPoint1[24615] = {X 458.4596, Y 50.7200, Z -2.1667, A 0.000, B 0.000, C 0.000 }
gfCNCPoint1[24616] = {X 475.0000, Y 50.7200, Z -2.1667, A 0.000, B 0.000, C 0.000 }
gfCNCPoint1[24617] = {X 476.0441, Y 50.7953, Z -2.1667, A 0.000, B 0.000, C 0.000 }
gfCNCPoint1[24618] = {X 477.0665, Y 51.0195, Z -2.1667, A 0.000, B 0.000, C 0.000 }
gfCNCPoint1[24619] = {X 478.0463, Y 51.3880, Z -2.1667, A 0.000, B 0.000, C 0.000 }
gfCNCPoint1[24620] = {X 478.9630, Y 51.8932, Z -2.1667, A 0.000, B 0.000, C 0.000 }
gfCNCPoint1[24621] = {X 479.9169, Y 52.6313, Z -2.1667, A 0.000, B 0.000, C 0.000 }
gfCNCPoint1[24622] = {X 480.7358, Y 53.5168, Z -2.1667, A 0.000, B 0.000, C 0.000 }
gfCNCPoint1[24623] = {X 481.3972, Y 54.5253, Z -2.1667, A 0.000, B 0.000, C 0.000 }
gfCNCPoint1[24624] = {X 481.8831, Y 55.6291, Z -2.1667, A 0.000, B 0.000, C 0.000 }
gfCNCPoint1[24625] = {X 482.1801, Y 56.7981, Z -2.1667, A 0.000, B 0.000, C 0.000 }
gfCNCPoint1[24626] = {X 482.2800, Y 58.0000, Z -2.1667, A 0.000, B 0.000, C 0.000 }
gfCNCPoint1[24627] = {X 482.2798, Y 58.9942, Z -2.1667, A 0.000, B 0.000, C 0.000 }
gfCNCPoint1[24628] = {X 482.1577, Y 60.2627, Z -2.1667, A 0.000, B 0.000, C 0.000 }
gfCNCPoint1[24629] = {X 481.8164, Y 61.4905, Z -2.1667, A 0.000, B 0.000, C 0.000 }
gfCNCPoint1[24630] = {X 481.2661, Y 62.6400, Z -2.1667, A 0.000, B 0.000, C 0.000 }
gfCNCPoint1[24631] = {X 480.5239, Y 63.6759, Z -2.1667, A 0.000, B 0.000, C 0.000 }
gfCNCPoint1[24632] = {X 479.6124, Y 64.5665, Z -2.1667, A 0.000, B 0.000, C 0.000 }
gfCNCPoint1[24633] = {X 478.5595, Y 65.2845, Z -2.1667, A 0.000, B 0.000, C 0.000 }
gfCNCPoint1[24634] = {X 478.5599, Y 90.7250, Z -2.1667, A 0.000, B 0.000, C 0.000 }
gfCNCPoint1[24635] = {X 479.5424, Y 91.3835, Z -2.1667, A 0.000, B 0.000, C 0.000 }
gfCNCPoint1[24636] = {X 480.4048, Y 92.1929, Z -2.1667, A 0.000, B 0.000, C 0.000 }
gfCNCPoint1[24637] = {X 481.1243, Y 93.1317, Z -2.1667, A 0.000, B 0.000, C 0.000 }
gfCNCPoint1[24638] = {X 481.6816, Y 94.1750, Z -2.1667, A 0.000, B 0.000, C 0.000 }
gfCNCPoint1[24639] = {X 482.0620, Y 95.2949, Z -2.1667, A 0.000, B 0.000, C 0.000 }
gfCNCPoint1[24640] = {X 507.6819, Y 95.2949, Z -2.1667, A 0.000, B 0.000, C 0.000 }
gfCNCPoint1[24641] = {X 507.6819, Y 97.6949, Z -2.1667, A 0.000, B 0.000, C 0.000 }
gfCNCPoint1[24642] = {X 597.6965, Y 97.6949, Z -2.1667, A 0.000, B 0.000, C 0.000 }
gfCNCPoint1[24643] = {X 597.6965, Y 51.8000, Z -2.1667, A 0.000, B 0.000, C 0.000 }
gfCNCPoint1[24644] = {X 593.5565, Y 51.8000, Z -2.1667, A 0.000, B 0.000, C 0.000 }
gfCNCPoint1[24645] = {X 592.3428, Y 51.6908, Z -2.1667, A 0.000, B 0.000, C 0.000 }
gfCNCPoint1[24646] = {X 591.1680, Y 51.3667, Z -2.1667, A 0.000, B 0.000, C 0.000 }
gfCNCPoint1[24647] = {X 590.0699, Y 50.8381, Z -2.1667, A 0.000, B 0.000, C 0.000 }
gfCNCPoint1[24648] = {X 589.0838, Y 50.1220, Z -2.1667, A 0.000, B 0.000, C 0.000 }
gfCNCPoint1[24649] = {X 588.4736, Y 49.5171, Z -2.1667, A 0.000, B 0.000, C 0.000 }
gfCNCPoint1[24650] = {X 587.9446, Y 48.8401, Z -2.1667, A 0.000, B 0.000, C 0.000 }
gfCNCPoint1[24651] = {X 587.5052, Y 48.1018, Z -2.1667, A 0.000, B 0.000, C 0.000 }
gfCNCPoint1[24652] = {X 587.0658, Y 48.8401, Z -2.1667, A 0.000, B 0.000, C 0.000 }
gfCNCPoint1[24653] = {X 586.5368, Y 49.5171, Z -2.1667, A 0.000, B 0.000, C 0.000 }
gfCNCPoint1[24654] = {X 585.9266, Y 50.1220, Z -2.1667, A 0.000, B 0.000, C 0.000 }
gfCNCPoint1[24655] = {X 585.1803, Y 50.6880, Z -2.1667, A 0.000, B 0.000, C 0.000 }
gfCNCPoint1[24656] = {X 584.3634, Y 51.1461, Z -2.1667, A 0.000, B 0.000, C 0.000 }
gfCNCPoint1[24657] = {X 583.3013, Y 51.5442, Z -2.1667, A 0.000, B 0.000, C 0.000 }
gfCNCPoint1[24658] = {X 582.1877, Y 51.7603, Z -2.1667, A 0.000, B 0.000, C 0.000 }
gfCNCPoint1[24659] = {X 581.0538, Y 51.7882, Z -2.1667, A 0.000, B 0.000, C 0.000 }
gfCNCPoint1[24660] = {X 579.9310, Y 51.6273, Z -2.1667, A 0.000, B 0.000, C 0.000 }
gfCNCPoint1[24661] = {X 578.8505, Y 51.2819, Z -2.1667, A 0.000, B 0.000, C 0.000 }
gfCNCPoint1[24662] = {X 577.8425, Y 50.7618, Z -2.1667, A 0.000, B 0.000, C 0.000 }
gfCNCPoint1[24663] = {X 576.9350, Y 50.0813, Z -2.1667, A 0.000, B 0.000, C 0.000 }
gfCNCPoint1[24664] = {X 576.3133, Y 49.4513, Z -2.1667, A 0.000, B 0.000, C 0.000 }
gfCNCPoint1[24665] = {X 575.7786, Y 48.7459, Z -2.1667, A 0.000, B 0.000, C 0.000 }
gfCNCPoint1[24666] = {X 575.3401, Y 47.9770, Z -2.1667, A 0.000, B 0.000, C 0.000 }
gfCNCPoint1[24667] = {X 574.9017, Y 48.7459, Z -2.1667, A 0.000, B 0.000, C 0.000 }
gfCNCPoint1[24668] = {X 574.3670, Y 49.4513, Z -2.1667, A 0.000, B 0.000, C 0.000 }
gfCNCPoint1[24669] = {X 573.7453, Y 50.0813, Z -2.1667, A 0.000, B 0.000, C 0.000 }
gfCNCPoint1[24670] = {X 572.7526, Y 50.8143, Z -2.1667, A 0.000, B 0.000, C 0.000 }
gfCNCPoint1[24671] = {X 571.6437, Y 51.3558, Z -2.1667, A 0.000, B 0.000, C 0.000 }
gfCNCPoint1[24672] = {X 570.4553, Y 51.6880, Z -2.1667, A 0.000, B 0.000, C 0.000 }
gfCNCPoint1[24673] = {X 569.2264, Y 51.8000, Z -2.1667, A 0.000, B 0.000, C 0.000 }
gfCNCPoint1[24674] = {X 562.4443, Y 51.8000, Z -2.1667, A 0.000, B 0.000, C 0.000 }
gfCNCPoint1[24675] = {X 561.2635, Y 51.6967, Z -2.1667, A 0.000, B 0.000, C 0.000 }
gfCNCPoint1[24676] = {X 560.1186, Y 51.3899, Z -2.1667, A 0.000, B 0.000, C 0.000 }
gfCNCPoint1[24677] = {X 559.0443, Y 50.8890, Z -2.1667, A 0.000, B 0.000, C 0.000 }
gfCNCPoint1[24678] = {X 558.0733, Y 50.2091, Z -2.1667, A 0.000, B 0.000, C 0.000 }
gfCNCPoint1[24679] = {X 557.2352, Y 49.3710, Z -2.1667, A 0.000, B 0.000, C 0.000 }
gfCNCPoint1[24680] = {X 556.5553, Y 48.4000, Z -2.1667, A 0.000, B 0.000, C 0.000 }
gfCNCPoint1[24681] = {X 556.0544, Y 47.3257, Z -2.1667, A 0.000, B 0.000, C 0.000 }
gfCNCPoint1[24682] = {X 555.7476, Y 46.1808, Z -2.1667, A 0.000, B 0.000, C 0.000 }
gfCNCPoint1[24683] = {X 555.6443, Y 45.0000, Z -2.1667, A 0.000, B 0.000, C 0.000 }
gfCNCPoint1[24684] = {X 555.6443, Y 44.0661, Z -2.1667, A 0.000, B 0.000, C 0.000 }
gfCNCPoint1[24685] = {X 555.7458, Y 42.9114, Z -2.1667, A 0.000, B 0.000, C 0.000 }
gfCNCPoint1[24686] = {X 556.0409, Y 41.7905, Z -2.1667, A 0.000, B 0.000, C 0.000 }
gfCNCPoint1[24687] = {X 556.5212, Y 40.7355, Z -2.1667, A 0.000, B 0.000, C 0.000 }
gfCNCPoint1[24688] = {X 557.1727, Y 39.7768, Z -2.1667, A 0.000, B 0.000, C 0.000 }
gfCNCPoint1[24689] = {X 557.1727, Y 10.2294, Z -2.1667, A 0.000, B 0.000, C 0.000 }
gfCNCPoint1[24690] = {X 556.5262, Y 9.2831, Z -2.1667, A 0.000, B 0.000, C 0.000 }
gfCNCPoint1[24691] = {X 556.0478, Y 8.2417, Z -2.1667, A 0.000, B 0.000, C 0.000 }
gfCNCPoint1[24692] = {X 555.7512, Y 7.1348, Z -2.1667, A 0.000, B 0.000, C 0.000 }
gfCNCPoint1[24693] = {X 555.6446, Y 5.9937, Z -2.1667, A 0.000, B 0.000, C 0.000 }
gfCNCPoint1[24694] = {X 555.6443, Y 5.0000, Z -2.1667, A 0.000, B 0.000, C 0.000 }
gfCNCPoint1[24695] = {X 555.6452, Y 4.8910, Z -2.1667, A 0.000, B 0.000, C 0.000 }
gfCNCPoint1[24696] = {X 555.6478, Y 4.7820, Z -2.1667, A 0.000, B 0.000, C 0.000 }
gfCNCPoint1[24697] = {X 555.8079, Y 3.5175, Z -2.1667, A 0.000, B 0.000, C 0.000 }
gfCNCPoint1[24698] = {X 556.2011, Y 2.3051, Z -2.1667, A 0.000, B 0.000, C 0.000 }
gfCNCPoint1[24699] = {X 358.2576, Y 2.3051, Z -2.1667, A 0.000, B 0.000, C 0.000 }
gfCNCPoint1[24700] = {X 360.1191, Y 3.4748, Z -2.1667, A 0.000, B 0.000, C 0.000 }
gfCNCPoint1[24701] = {X 361.8521, Y 4.8277, Z -2.1667, A 0.000, B 0.000, C 0.000 }
gfCNCPoint1[24702] = {X 363.4384, Y 6.3499, Z -2.1667, A 0.000, B 0.000, C 0.000 }
gfCNCPoint1[24703] = {X 363.7836, Y 6.7255, Z -2.1667, A 0.000, B 0.000, C 0.000 }
gfCNCPoint1[24704] = {X 364.1198, Y 7.1091, Z -2.1667, A 0.000, B 0.000, C 0.000 }
gfCNCPoint1[24705] = {X 365.6217, Y 9.0473, Z -2.1667, A 0.000, B 0.000, C 0.000 }
gfCNCPoint1[24706] = {X 366.9287, Y 11.1217, Z -2.1667, A 0.000, B 0.000, C 0.000 }
gfCNCPoint1[24707] = {X 368.0285, Y 13.3131, Z -2.1667, A 0.000, B 0.000, C 0.000 }
gfCNCPoint1[24708] = {X 368.9110, Y 15.6007, Z -2.1667, A 0.000, B 0.000, C 0.000 }
gfCNCPoint1[24709] = {X 369.5676, Y 17.9630, Z -2.1667, A 0.000, B 0.000, C 0.000 }
gfCNCPoint1[24710] = {X 370.0560, Y 20.6425, Z -2.1667, A 0.000, B 0.000, C 0.000 }
gfCNCPoint1[24711] = {X 370.3161, Y 23.3536, Z -2.1667, A 0.000, B 0.000, C 0.000 }
gfCNCPoint1[24712] = {X 370.3462, Y 26.0770, Z -2.1667, A 0.000, B 0.000, C 0.000 }
gfCNCPoint1[24713] = {X 370.1459, Y 28.7932, Z -2.1667, A 0.000, B 0.000, C 0.000 }
gfCNCPoint1[24714] = {X 369.7168, Y 31.4827, Z -2.1667, A 0.000, B 0.000, C 0.000 }
gfCNCPoint1[24715] = {X 369.1810, Y 33.6350, Z -2.1667, A 0.000, B 0.000, C 0.000 }
gfCNCPoint1[24716] = {X 368.4572, Y 35.7315, Z -2.1667, A 0.000, B 0.000, C 0.000 }
gfCNCPoint1[24717] = {X 367.5509, Y 37.7559, Z -2.1667, A 0.000, B 0.000, C 0.000 }
gfCNCPoint1[24718] = {X 366.4692, Y 39.6923, Z -2.1667, A 0.000, B 0.000, C 0.000 }
gfCNCPoint1[24719] = {X 365.2207, Y 41.5255, Z -2.1667, A 0.000, B 0.000, C 0.000 }
gfCNCPoint1[24720] = {X 363.9632, Y 43.0749, Z -2.1667, A 0.000, B 0.000, C 0.000 }
gfCNCPoint1[24721] = {X 362.5748, Y 44.5082, Z -2.1667, A 0.000, B 0.000, C 0.000 }
gfCNCPoint1[24722] = {X 361.0660, Y 45.8143, Z -2.1667, A 0.000, B 0.000, C 0.000 }
gfCNCPoint1[24723] = {X 359.4485, Y 46.9830, Z -2.1667, A 0.000, B 0.000, C 0.000 }
gfCNCPoint1[24724] = {X 357.7348, Y 48.0055, Z -2.1667, A 0.000, B 0.000, C 0.000 }
gfCNCPoint1[24725] = {X 355.7251, Y 48.9197, Z -2.1667, A 0.000, B 0.000, C 0.000 }
gfCNCPoint1[24726] = {X 353.6376, Y 49.6386, Z -2.1667, A 0.000, B 0.000, C 0.000 }
gfCNCPoint1[24727] = {X 351.4911, Y 50.1558, Z -2.1667, A 0.000, B 0.000, C 0.000 }
gfCNCPoint1[24728] = {X 349.3053, Y 50.4665, Z -2.1667, A 0.000, B 0.000, C 0.000 }
gfCNCPoint1[24729] = {X 347.0997, Y 50.5679, Z -2.1667, A 0.000, B 0.000, C 0.000 }
gfCNCPoint1[24730] = {X 344.9865, Y 50.5317, Z -2.1667, A 0.000, B 0.000, C 0.000 }
gfCNCPoint1[24731] = {X 342.8843, Y 50.3124, Z -2.1667, A 0.000, B 0.000, C 0.000 }
gfCNCPoint1[24732] = {X 340.8090, Y 49.9118, Z -2.1667, A 0.000, B 0.000, C 0.000 }
gfCNCPoint1[24733] = {X 338.7763, Y 49.3329, Z -2.1667, A 0.000, B 0.000, C 0.000 }
gfCNCPoint1[24734] = {X 336.8014, Y 48.5800, Z -2.1667, A 0.000, B 0.000, C 0.000 }
gfCNCPoint1[24735] = {X 334.8991, Y 47.6588, Z -2.1667, A 0.000, B 0.000, C 0.000 }
gfCNCPoint1[24736] = {X 333.3430, Y 46.7016, Z -2.1667, A 0.000, B 0.000, C 0.000 }
gfCNCPoint1[24737] = {X 331.8620, Y 45.6317, Z -2.1667, A 0.000, B 0.000, C 0.000 }
gfCNCPoint1[24738] = {X 330.4645, Y 44.4549, Z -2.1667, A 0.000, B 0.000, C 0.000 }
gfCNCPoint1[24739] = {X 329.4670, Y 44.4079, Z -2.1667, A 0.000, B 0.000, C 0.000 }
gfCNCPoint1[24740] = {X 328.5000, Y 44.1589, Z -2.1667, A 0.000, B 0.000, C 0.000 }
gfCNCPoint1[24741] = {X 327.6040, Y 43.7182, Z -2.1667, A 0.000, B 0.000, C 0.000 }
gfCNCPoint1[24742] = {X 326.8164, Y 43.1044, Z -2.1667, A 0.000, B 0.000, C 0.000 }
gfCNCPoint1[24743] = {X 326.1897, Y 42.4934, Z -2.1667, A 0.000, B 0.000, C 0.000 }
gfCNCPoint1[24744] = {X 325.5686, Y 41.7541, Z -2.1667, A 0.000, B 0.000, C 0.000 }
gfCNCPoint1[24745] = {X 325.1052, Y 40.9070, Z -2.1667, A 0.000, B 0.000, C 0.000 }
gfCNCPoint1[24746] = {X 324.8177, Y 39.9852, Z -2.1667, A 0.000, B 0.000, C 0.000 }
gfCNCPoint1[24747] = {X 324.7172, Y 39.0249, Z -2.1667, A 0.000, B 0.000, C 0.000 }
gfCNCPoint1[24748] = {X 324.8079, Y 38.0635, Z -2.1667, A 0.000, B 0.000, C 0.000 }
gfCNCPoint1[24749] = {X 325.0860, Y 37.1389, Z -2.1667, A 0.000, B 0.000, C 0.000 }
gfCNCPoint1[24750] = {X 325.5408, Y 36.2871, Z -2.1667, A 0.000, B 0.000, C 0.000 }
gfCNCPoint1[24751] = {X 329.7765, Y 29.9538, Z -2.1667, A 0.000, B 0.000, C 0.000 }
gfCNCPoint1[24752] = {X 330.4614, Y 29.1399, Z -2.1667, A 0.000, B 0.000, C 0.000 }
gfCNCPoint1[24753] = {X 331.3063, Y 28.4938, Z -2.1667, A 0.000, B 0.000, C 0.000 }
gfCNCPoint1[24754] = {X 332.2712, Y 28.0462, Z -2.1667, A 0.000, B 0.000, C 0.000 }
gfCNCPoint1[24755] = {X 333.3101, Y 27.8182, Z -2.1667, A 0.000, B 0.000, C 0.000 }
gfCNCPoint1[24756] = {X 334.3738, Y 27.8207, Z -2.1667, A 0.000, B 0.000, C 0.000 }
gfCNCPoint1[24757] = {X 335.4116, Y 28.0536, Z -2.1667, A 0.000, B 0.000, C 0.000 }
gfCNCPoint1[24758] = {X 336.3743, Y 28.5058, Z -2.1667, A 0.000, B 0.000, C 0.000 }
gfCNCPoint1[24759] = {X 337.2162, Y 29.1559, Z -2.1667, A 0.000, B 0.000, C 0.000 }
gfCNCPoint1[24760] = {X 337.7863, Y 29.7052, Z -2.1667, A 0.000, B 0.000, C 0.000 }
gfCNCPoint1[24761] = {X 338.3566, Y 30.3621, Z -2.1667, A 0.000, B 0.000, C 0.000 }
gfCNCPoint1[24762] = {X 338.8011, Y 31.1098, Z -2.1667, A 0.000, B 0.000, C 0.000 }
gfCNCPoint1[24763] = {X 339.1058, Y 31.9246, Z -2.1667, A 0.000, B 0.000, C 0.000 }
gfCNCPoint1[24764] = {X 339.2610, Y 32.7805, Z -2.1667, A 0.000, B 0.000, C 0.000 }
gfCNCPoint1[24765] = {X 339.2618, Y 33.6504, Z -2.1667, A 0.000, B 0.000, C 0.000 }
gfCNCPoint1[24766] = {X 339.9060, Y 34.2218, Z -2.1667, A 0.000, B 0.000, C 0.000 }
gfCNCPoint1[24767] = {X 340.5746, Y 34.7645, Z -2.1667, A 0.000, B 0.000, C 0.000 }
gfCNCPoint1[24768] = {X 341.8064, Y 35.5733, Z -2.1667, A 0.000, B 0.000, C 0.000 }
gfCNCPoint1[24769] = {X 343.1432, Y 36.1933, Z -2.1667, A 0.000, B 0.000, C 0.000 }
gfCNCPoint1[24770] = {X 344.5562, Y 36.6113, Z -2.1667, A 0.000, B 0.000, C 0.000 }
gfCNCPoint1[24771] = {X 346.0151, Y 36.8183, Z -2.1667, A 0.000, B 0.000, C 0.000 }
gfCNCPoint1[24772] = {X 347.4887, Y 36.8099, Z -2.1667, A 0.000, B 0.000, C 0.000 }
gfCNCPoint1[24773] = {X 348.8410, Y 36.6281, Z -2.1667, A 0.000, B 0.000, C 0.000 }
gfCNCPoint1[24774] = {X 350.1456, Y 36.2281, Z -2.1667, A 0.000, B 0.000, C 0.000 }
gfCNCPoint1[24775] = {X 351.3675, Y 35.6207, Z -2.1667, A 0.000, B 0.000, C 0.000 }
gfCNCPoint1[24776] = {X 352.4739, Y 34.8221, Z -2.1667, A 0.000, B 0.000, C 0.000 }
gfCNCPoint1[24777] = {X 353.5724, Y 33.7525, Z -2.1667, A 0.000, B 0.000, C 0.000 }
gfCNCPoint1[24778] = {X 354.5233, Y 32.5496, Z -2.1667, A 0.000, B 0.000, C 0.000 }
gfCNCPoint1[24779] = {X 355.3104, Y 31.2339, Z -2.1667, A 0.000, B 0.000, C 0.000 }
gfCNCPoint1[24780] = {X 355.9206, Y 29.8273, Z -2.1667, A 0.000, B 0.000, C 0.000 }
gfCNCPoint1[24781] = {X 356.3436, Y 28.3536, Z -2.1667, A 0.000, B 0.000, C 0.000 }
gfCNCPoint1[24782] = {X 356.6081, Y 26.7184, Z -2.1667, A 0.000, B 0.000, C 0.000 }
gfCNCPoint1[24783] = {X 356.7158, Y 25.0656, Z -2.1667, A 0.000, B 0.000, C 0.000 }
gfCNCPoint1[24784] = {X 356.6657, Y 23.4100, Z -2.1667, A 0.000, B 0.000, C 0.000 }
gfCNCPoint1[24785] = {X 356.4583, Y 21.7667, Z -2.1667, A 0.000, B 0.000, C 0.000 }
gfCNCPoint1[24786] = {X 356.1379, Y 20.3836, Z -2.1667, A 0.000, B 0.000, C 0.000 }
gfCNCPoint1[24787] = {X 355.6487, Y 19.0509, Z -2.1667, A 0.000, B 0.000, C 0.000 }
gfCNCPoint1[24788] = {X 354.9983, Y 17.7891, Z -2.1667, A 0.000, B 0.000, C 0.000 }
gfCNCPoint1[24789] = {X 354.1966, Y 16.6175, Z -2.1667, A 0.000, B 0.000, C 0.000 }
gfCNCPoint1[24790] = {X 353.3644, Y 15.6890, Z -2.1667, A 0.000, B 0.000, C 0.000 }
gfCNCPoint1[24791] = {X 352.4077, Y 14.8892, Z -2.1667, A 0.000, B 0.000, C 0.000 }
gfCNCPoint1[24792] = {X 351.3464, Y 14.2349, Z -2.1667, A 0.000, B 0.000, C 0.000 }
gfCNCPoint1[24793] = {X 350.2022, Y 13.7393, Z -2.1667, A 0.000, B 0.000, C 0.000 }
gfCNCPoint1[24794] = {X 348.9988, Y 13.4128, Z -2.1667, A 0.000, B 0.000, C 0.000 }
gfCNCPoint1[24795] = {X 347.3616, Y 13.2061, Z -2.1667, A 0.000, B 0.000, C 0.000 }
gfCNCPoint1[24796] = {X 345.7113, Y 13.2115, Z -2.1667, A 0.000, B 0.000, C 0.000 }
gfCNCPoint1[24797] = {X 344.0755, Y 13.4287, Z -2.1667, A 0.000, B 0.000, C 0.000 }
gfCNCPoint1[24798] = {X 342.4810, Y 13.8542, Z -2.1667, A 0.000, B 0.000, C 0.000 }
gfCNCPoint1[24799] = {X 340.9544, Y 14.4809, Z -2.1667, A 0.000, B 0.000, C 0.000 }
gfCNCPoint1[24800] = {X 339.5210, Y 15.2984, Z -2.1667, A 0.000, B 0.000, C 0.000 }
gfCNCPoint1[24801] = {X 339.4274, Y 16.1844, Z -2.1667, A 0.000, B 0.000, C 0.000 }
gfCNCPoint1[24802] = {X 339.1742, Y 17.0386, Z -2.1667, A 0.000, B 0.000, C 0.000 }
gfCNCPoint1[24803] = {X 338.7701, Y 17.8325, Z -2.1667, A 0.000, B 0.000, C 0.000 }
gfCNCPoint1[24804] = {X 338.2283, Y 18.5397, Z -2.1667, A 0.000, B 0.000, C 0.000 }
gfCNCPoint1[24805] = {X 337.5670, Y 19.1366, Z -2.1667, A 0.000, B 0.000, C 0.000 }
gfCNCPoint1[24806] = {X 336.8400, Y 19.6716, Z -2.1667, A 0.000, B 0.000, C 0.000 }
gfCNCPoint1[24807] = {X 335.9171, Y 20.1909, Z -2.1667, A 0.000, B 0.000, C 0.000 }
gfCNCPoint1[24808] = {X 334.9039, Y 20.4988, Z -2.1667, A 0.000, B 0.000, C 0.000 }
gfCNCPoint1[24809] = {X 333.8481, Y 20.5809, Z -2.1667, A 0.000, B 0.000, C 0.000 }
gfCNCPoint1[24810] = {X 332.7995, Y 20.4334, Z -2.1667, A 0.000, B 0.000, C 0.000 }
gfCNCPoint1[24811] = {X 331.8074, Y 20.0631, Z -2.1667, A 0.000, B 0.000, C 0.000 }
gfCNCPoint1[24812] = {X 330.9186, Y 19.4876, Z -2.1667, A 0.000, B 0.000, C 0.000 }
gfCNCPoint1[24813] = {X 330.1748, Y 18.7338, Z -2.1667, A 0.000, B 0.000, C 0.000 }
gfCNCPoint1[24814] = {X 329.6111, Y 17.8373, Z -2.1667, A 0.000, B 0.000, C 0.000 }
gfCNCPoint1[24815] = {X 326.0906, Y 10.5950, Z -2.1667, A 0.000, B 0.000, C 0.000 }
gfCNCPoint1[24816] = {X 325.7555, Y 9.6856, Z -2.1667, A 0.000, B 0.000, C 0.000 }
gfCNCPoint1[24817] = {X 325.6067, Y 8.7279, Z -2.1667, A 0.000, B 0.000, C 0.000 }
gfCNCPoint1[24818] = {X 325.6502, Y 7.7597, Z -2.1667, A 0.000, B 0.000, C 0.000 }
gfCNCPoint1[24819] = {X 325.8841, Y 6.8192, Z -2.1667, A 0.000, B 0.000, C 0.000 }
gfCNCPoint1[24820] = {X 326.2993, Y 5.9435, Z -2.1667, A 0.000, B 0.000, C 0.000 }
gfCNCPoint1[24821] = {X 326.9294, Y 5.1132, Z -2.1667, A 0.000, B 0.000, C 0.000 }
gfCNCPoint1[24822] = {X 327.7213, Y 4.4357, Z -2.1667, A 0.000, B 0.000, C 0.000 }
gfCNCPoint1[24823] = {X 328.3968, Y 3.9733, Z -2.1667, A 0.000, B 0.000, C 0.000 }
gfCNCPoint1[24824] = {X 329.3297, Y 3.4827, Z -2.1667, A 0.000, B 0.000, C 0.000 }
gfCNCPoint1[24825] = {X 330.3462, Y 3.2039, Z -2.1667, A 0.000, B 0.000, C 0.000 }
gfCNCPoint1[24826] = {X 331.3989, Y 3.1499, Z -2.1667, A 0.000, B 0.000, C 0.000 }
gfCNCPoint1[24827] = {X 332.4386, Y 3.3232, Z -2.1667, A 0.000, B 0.000, C 0.000 }
gfCNCPoint1[24828] = {X 333.3762, Y 2.7965, Z -2.1667, A 0.000, B 0.000, C 0.000 }
gfCNCPoint1[24829] = {X 334.3328, Y 2.3051, Z -2.1667, A 0.000, B 0.000, C 0.000 }
gfCNCPoint1[24830] = {X 334.5442, Y 2.7360, Z -2.1667, A 0.000, B 0.000, C 0.000 }
gfCNCPoint1[24831] = {X 335.0201, Y 2.5081, Z -2.1667, A 0.000, B 0.000, C 0.000 }
gfCNCPoint1[24832] = {X 335.5002, Y 2.2890, Z -2.1667, A 0.000, B 0.000, C 0.000 }
gfCNCPoint1[24833] = {X 335.8480, Y 2.1341, Z -2.1667, A 0.000, B 0.000, C 0.000 }
gfCNCPoint1[24834] = {X 337.9511, Y 1.3136, Z -2.1667, A 0.000, B 0.000, C 0.000 }
gfCNCPoint1[24835] = {X 340.1168, Y 0.6761, Z -2.1667, A 0.000, B 0.000, C 0.000 }
gfCNCPoint1[24836] = {X 342.3290, Y 0.2262, Z -2.1667, A 0.000, B 0.000, C 0.000 }
gfCNCPoint1[24837] = {X 344.5717, Y -0.0328, Z -2.1667, A 0.000, B 0.000, C 0.000 }
gfCNCPoint1[24838] = {X 346.8282, Y -0.0989, Z -2.1667, A 0.000, B 0.000, C 0.000 }
gfCNCPoint1[24839] = {X 349.0822, Y 0.0282, Z -2.1667, A 0.000, B 0.000, C 0.000 }
gfCNCPoint1[24840] = {X 351.3170, Y 0.3478, Z -2.1667, A 0.000, B 0.000, C 0.000 }
gfCNCPoint1[24841] = {X 351.8871, Y 0.4533, Z -2.1667, A 0.000, B 0.000, C 0.000 }
gfCNCPoint1[24842] = {X 353.8286, Y 0.9413, Z -2.1667, A 0.000, B 0.000, C 0.000 }
gfCNCPoint1[24843] = {X 355.7152, Y 1.6110, Z -2.1667, A 0.000, B 0.000, C 0.000 }
gfCNCPoint1[24844] = {X 357.5298, Y 2.4565, Z -2.1667, A 0.000, B 0.000, C 0.000 }
gfCNCPoint1[24845] = {X 359.2561, Y 3.4701, Z -2.1667, A 0.000, B 0.000, C 0.000 }
gfCNCPoint1[24846] = {X 360.8787, Y 4.6426, Z -2.1667, A 0.000, B 0.000, C 0.000 }
gfCNCPoint1[24847] = {X 362.3829, Y 5.9636, Z -2.1667, A 0.000, B 0.000, C 0.000 }
gfCNCPoint1[24848] = {X 363.7552, Y 7.4212, Z -2.1667, A 0.000, B 0.000, C 0.000 }
gfCNCPoint1[24849] = {X 365.2285, Y 9.3225, Z -2.1667, A 0.000, B 0.000, C 0.000 }
gfCNCPoint1[24850] = {X 366.5106, Y 11.3576, Z -2.1667, A 0.000, B 0.000, C 0.000 }
gfCNCPoint1[24851] = {X 367.5896, Y 13.5074, Z -2.1667, A 0.000, B 0.000, C 0.000 }
gfCNCPoint1[24852] = {X 368.4553, Y 15.7515, Z -2.1667, A 0.000, B 0.000, C 0.000 }
gfCNCPoint1[24853] = {X 369.0994, Y 18.0690, Z -2.1667, A 0.000, B 0.000, C 0.000 }
gfCNCPoint1[24854] = {X 369.5805, Y 20.7085, Z -2.1667, A 0.000, B 0.000, C 0.000 }
gfCNCPoint1[24855] = {X 369.8368, Y 23.3792, Z -2.1667, A 0.000, B 0.000, C 0.000 }
gfCNCPoint1[24856] = {X 369.8664, Y 26.0620, Z -2.1667, A 0.000, B 0.000, C 0.000 }
gfCNCPoint1[24857] = {X 369.6691, Y 28.7377, Z -2.1667, A 0.000, B 0.000, C 0.000 }
gfCNCPoint1[24858] = {X 369.2464, Y 31.3871, Z -2.1667, A 0.000, B 0.000, C 0.000 }
gfCNCPoint1[24859] = {X 368.7208, Y 33.4985, Z -2.1667, A 0.000, B 0.000, C 0.000 }
gfCNCPoint1[24860] = {X 368.0108, Y 35.5551, Z -2.1667, A 0.000, B 0.000, C 0.000 }
gfCNCPoint1[24861] = {X 367.1217, Y 37.5410, Z -2.1667, A 0.000, B 0.000, C 0.000 }
gfCNCPoint1[24862] = {X 366.0606, Y 39.4405, Z -2.1667, A 0.000, B 0.000, C 0.000 }
gfCNCPoint1[24863] = {X 364.8357, Y 41.2388, Z -2.1667, A 0.000, B 0.000, C 0.000 }
gfCNCPoint1[24864] = {X 363.6036, Y 42.7570, Z -2.1667, A 0.000, B 0.000, C 0.000 }
gfCNCPoint1[24865] = {X 362.2431, Y 44.1612, Z -2.1667, A 0.000, B 0.000, C 0.000 }
gfCNCPoint1[24866] = {X 360.7645, Y 45.4406, Z -2.1667, A 0.000, B 0.000, C 0.000 }
gfCNCPoint1[24867] = {X 359.1794, Y 46.5854, Z -2.1667, A 0.000, B 0.000, C 0.000 }
gfCNCPoint1[24868] = {X 357.5000, Y 47.5867, Z -2.1667, A 0.000, B 0.000, C 0.000 }
gfCNCPoint1[24869] = {X 355.5332, Y 48.4796, Z -2.1667, A 0.000, B 0.000, C 0.000 }
gfCNCPoint1[24870] = {X 353.4904, Y 49.1816, Z -2.1667, A 0.000, B 0.000, C 0.000 }
gfCNCPoint1[24871] = {X 351.3903, Y 49.6864, Z -2.1667, A 0.000, B 0.000, C 0.000 }
gfCNCPoint1[24872] = {X 349.2516, Y 49.9894, Z -2.1667, A 0.000, B 0.000, C 0.000 }
gfCNCPoint1[24873] = {X 347.0938, Y 50.0879, Z -2.1667, A 0.000, B 0.000, C 0.000 }
gfCNCPoint1[24874] = {X 345.0197, Y 50.0528, Z -2.1667, A 0.000, B 0.000, C 0.000 }
gfCNCPoint1[24875] = {X 342.9564, Y 49.8379, Z -2.1667, A 0.000, B 0.000, C 0.000 }
gfCNCPoint1[24876] = {X 340.9196, Y 49.4447, Z -2.1667, A 0.000, B 0.000, C 0.000 }
gfCNCPoint1[24877] = {X 338.9246, Y 48.8763, Z -2.1667, A 0.000, B 0.000, C 0.000 }
gfCNCPoint1[24878] = {X 336.9864, Y 48.1370, Z -2.1667, A 0.000, B 0.000, C 0.000 }
gfCNCPoint1[24879] = {X 335.1196, Y 47.2323, Z -2.1667, A 0.000, B 0.000, C 0.000 }
gfCNCPoint1[24880] = {X 333.5424, Y 46.2576, Z -2.1667, A 0.000, B 0.000, C 0.000 }
gfCNCPoint1[24881] = {X 332.0445, Y 45.1648, Z -2.1667, A 0.000, B 0.000, C 0.000 }
gfCNCPoint1[24882] = {X 330.6350, Y 43.9603, Z -2.1667, A 0.000, B 0.000, C 0.000 }
gfCNCPoint1[24883] = {X 329.6763, Y 43.9518, Z -2.1667, A 0.000, B 0.000, C 0.000 }
gfCNCPoint1[24884] = {X 328.7422, Y 43.7359, Z -2.1667, A 0.000, B 0.000, C 0.000 }
gfCNCPoint1[24885] = {X 327.8771, Y 43.3228, Z -2.1667, A 0.000, B 0.000, C 0.000 }
gfCNCPoint1[24886] = {X 327.1219, Y 42.7321, Z -2.1667, A 0.000, B 0.000, C 0.000 }
gfCNCPoint1[24887] = {X 326.5249, Y 42.1498, Z -2.1667, A 0.000, B 0.000, C 0.000 }
gfCNCPoint1[24888] = {X 325.8848, Y 41.3619, Z -2.1667, A 0.000, B 0.000, C 0.000 }
gfCNCPoint1[24889] = {X 325.4424, Y 40.4483, Z -2.1667, A 0.000, B 0.000, C 0.000 }
gfCNCPoint1[24890] = {X 325.2210, Y 39.4576, Z -2.1667, A 0.000, B 0.000, C 0.000 }
gfCNCPoint1[24891] = {X 325.2326, Y 38.4426, Z -2.1667, A 0.000, B 0.000, C 0.000 }
gfCNCPoint1[24892] = {X 325.4765, Y 37.4572, Z -2.1667, A 0.000, B 0.000, C 0.000 }
gfCNCPoint1[24893] = {X 325.9397, Y 36.5539, Z -2.1667, A 0.000, B 0.000, C 0.000 }
gfCNCPoint1[24894] = {X 330.1988, Y 30.1861, Z -2.1667, A 0.000, B 0.000, C 0.000 }
gfCNCPoint1[24895] = {X 330.8195, Y 29.4619, Z -2.1667, A 0.000, B 0.000, C 0.000 }
gfCNCPoint1[24896] = {X 331.5816, Y 28.8884, Z -2.1667, A 0.000, B 0.000, C 0.000 }
gfCNCPoint1[24897] = {X 332.4495, Y 28.4927, Z -2.1667, A 0.000, B 0.000, C 0.000 }
gfCNCPoint1[24898] = {X 333.3822, Y 28.2932, Z -2.1667, A 0.000, B 0.000, C 0.000 }
gfCNCPoint1[24899] = {X 334.3360, Y 28.2995, Z -2.1667, A 0.000, B 0.000, C 0.000 }
gfCNCPoint1[24900] = {X 335.2660, Y 28.5111, Z -2.1667, A 0.000, B 0.000, C 0.000 }
gfCNCPoint1[24901] = {X 336.1286, Y 28.9182, Z -2.1667, A 0.000, B 0.000, C 0.000 }
gfCNCPoint1[24902] = {X 336.8832, Y 29.5016, Z -2.1667, A 0.000, B 0.000, C 0.000 }
gfCNCPoint1[24903] = {X 337.4845, Y 30.0811, Z -2.1667, A 0.000, B 0.000, C 0.000 }
gfCNCPoint1[24904] = {X 338.1274, Y 30.8804, Z -2.1667, A 0.000, B 0.000, C 0.000 }
gfCNCPoint1[24905] = {X 338.5678, Y 31.8068, Z -2.1667, A 0.000, B 0.000, C 0.000 }
gfCNCPoint1[24906] = {X 338.7817, Y 32.8099, Z -2.1667, A 0.000, B 0.000, C 0.000 }
gfCNCPoint1[24907] = {X 338.7575, Y 33.8354, Z -2.1667, A 0.000, B 0.000, C 0.000 }
gfCNCPoint1[24908] = {X 339.5032, Y 34.5090, Z -2.1667, A 0.000, B 0.000, C 0.000 }
gfCNCPoint1[24909] = {X 340.2815, Y 35.1446, Z -2.1667, A 0.000, B 0.000, C 0.000 }
gfCNCPoint1[24910] = {X 341.4928, Y 35.9470, Z -2.1667, A 0.000, B 0.000, C 0.000 }
gfCNCPoint1[24911] = {X 342.8031, Y 36.5752, Z -2.1667, A 0.000, B 0.000, C 0.000 }
gfCNCPoint1[24912] = {X 344.1873, Y 37.0170, Z -2.1667, A 0.000, B 0.000, C 0.000 }
gfCNCPoint1[24913] = {X 345.6191, Y 37.2643, Z -2.1667, A 0.000, B 0.000, C 0.000 }
gfCNCPoint1[24914] = {X 347.0713, Y 37.3121, Z -2.1667, A 0.000, B 0.000, C 0.000 }
gfCNCPoint1[24915] = {X 347.5135, Y 37.2893, Z -2.1667, A 0.000, B 0.000, C 0.000 }
gfCNCPoint1[24916] = {X 348.9437, Y 37.0970, Z -2.1667, A 0.000, B 0.000, C 0.000 }
gfCNCPoint1[24917] = {X 350.3234, Y 36.6740, Z -2.1667, A 0.000, B 0.000, C 0.000 }
gfCNCPoint1[24918] = {X 351.6156, Y 36.0316, Z -2.1667, A 0.000, B 0.000, C 0.000 }
gfCNCPoint1[24919] = {X 352.7857, Y 35.1870, Z -2.1667, A 0.000, B 0.000, C 0.000 }
gfCNCPoint1[24920] = {X 353.9291, Y 34.0737, Z -2.1667, A 0.000, B 0.000, C 0.000 }
gfCNCPoint1[24921] = {X 354.9187, Y 32.8218, Z -2.1667, A 0.000, B 0.000, C 0.000 }
gfCNCPoint1[24922] = {X 355.7379, Y 31.4522, Z -2.1667, A 0.000, B 0.000, C 0.000 }
gfCNCPoint1[24923] = {X 356.3728, Y 29.9882, Z -2.1667, A 0.000, B 0.000, C 0.000 }
gfCNCPoint1[24924] = {X 356.8129, Y 28.4543, Z -2.1667, A 0.000, B 0.000, C 0.000 }
gfCNCPoint1[24925] = {X 357.0850, Y 26.7729, Z -2.1667, A 0.000, B 0.000, C 0.000 }
gfCNCPoint1[24926] = {X 357.1958, Y 25.0733, Z -2.1667, A 0.000, B 0.000, C 0.000 }
gfCNCPoint1[24927] = {X 357.1441, Y 23.3709, Z -2.1667, A 0.000, B 0.000, C 0.000 }
gfCNCPoint1[24928] = {X 356.9306, Y 21.6811, Z -2.1667, A 0.000, B 0.000, C 0.000 }
gfCNCPoint1[24929] = {X 356.5964, Y 20.2415, Z -2.1667, A 0.000, B 0.000, C 0.000 }
gfCNCPoint1[24930] = {X 356.0866, Y 18.8544, Z -2.1667, A 0.000, B 0.000, C 0.000 }
gfCNCPoint1[24931] = {X 355.4091, Y 17.5409, Z -2.1667, A 0.000, B 0.000, C 0.000 }
gfCNCPoint1[24932] = {X 354.5744, Y 16.3214, Z -2.1667, A 0.000, B 0.000, C 0.000 }
gfCNCPoint1[24933] = {X 353.6962, Y 15.3421, Z -2.1667, A 0.000, B 0.000, C 0.000 }
gfCNCPoint1[24934] = {X 352.6867, Y 14.4987, Z -2.1667, A 0.000, B 0.000, C 0.000 }
gfCNCPoint1[24935] = {X 351.5669, Y 13.8085, Z -2.1667, A 0.000, B 0.000, C 0.000 }
gfCNCPoint1[24936] = {X 350.3597, Y 13.2859, Z -2.1667, A 0.000, B 0.000, C 0.000 }
gfCNCPoint1[24937] = {X 349.0902, Y 12.9415, Z -2.1667, A 0.000, B 0.000, C 0.000 }
gfCNCPoint1[24938] = {X 347.3476, Y 12.7244, Z -2.1667, A 0.000, B 0.000, C 0.000 }
gfCNCPoint1[24939] = {X 345.5915, Y 12.7388, Z -2.1667, A 0.000, B 0.000, C 0.000 }
gfCNCPoint1[24940] = {X 343.8527, Y 12.9843, Z -2.1667, A 0.000, B 0.000, C 0.000 }
gfCNCPoint1[24941] = {X 342.1613, Y 13.4566, Z -2.1667, A 0.000, B 0.000, C 0.000 }
gfCNCPoint1[24942] = {X 340.5469, Y 14.1477, Z -2.1667, A 0.000, B 0.000, C 0.000 }
gfCNCPoint1[24943] = {X 339.0375, Y 15.0453, Z -2.1667, A 0.000, B 0.000, C 0.000 }
gfCNCPoint1[24944] = {X 338.9897, Y 15.9035, Z -2.1667, A 0.000, B 0.000, C 0.000 }
gfCNCPoint1[24945] = {X 338.7760, Y 16.7360, Z -2.1667, A 0.000, B 0.000, C 0.000 }
gfCNCPoint1[24946] = {X 338.4045, Y 17.5110, Z -2.1667, A 0.000, B 0.000, C 0.000 }
gfCNCPoint1[24947] = {X 337.8894, Y 18.1991, Z -2.1667, A 0.000, B 0.000, C 0.000 }
gfCNCPoint1[24948] = {X 337.2504, Y 18.7738, Z -2.1667, A 0.000, B 0.000, C 0.000 }
gfCNCPoint1[24949] = {X 336.5606, Y 19.2813, Z -2.1667, A 0.000, B 0.000, C 0.000 }
gfCNCPoint1[24950] = {X 335.7284, Y 19.7495, Z -2.1667, A 0.000, B 0.000, C 0.000 }
gfCNCPoint1[24951] = {X 334.8148, Y 20.0271, Z -2.1667, A 0.000, B 0.000, C 0.000 }
gfCNCPoint1[24952] = {X 333.8628, Y 20.1012, Z -2.1667, A 0.000, B 0.000, C 0.000 }
gfCNCPoint1[24953] = {X 332.9173, Y 19.9681, Z -2.1667, A 0.000, B 0.000, C 0.000 }
gfCNCPoint1[24954] = {X 332.0228, Y 19.6341, Z -2.1667, A 0.000, B 0.000, C 0.000 }
gfCNCPoint1[24955] = {X 331.2213, Y 19.1151, Z -2.1667, A 0.000, B 0.000, C 0.000 }
gfCNCPoint1[24956] = {X 330.5507, Y 18.4353, Z -2.1667, A 0.000, B 0.000, C 0.000 }
gfCNCPoint1[24957] = {X 330.0425, Y 17.6269, Z -2.1667, A 0.000, B 0.000, C 0.000 }
gfCNCPoint1[24958] = {X 326.5223, Y 10.3852, Z -2.1667, A 0.000, B 0.000, C 0.000 }
gfCNCPoint1[24959] = {X 326.2154, Y 9.5469, Z -2.1667, A 0.000, B 0.000, C 0.000 }
gfCNCPoint1[24960] = {X 326.0841, Y 8.6639, Z -2.1667, A 0.000, B 0.000, C 0.000 }
gfCNCPoint1[24961] = {X 326.1337, Y 7.7726, Z -2.1667, A 0.000, B 0.000, C 0.000 }
gfCNCPoint1[24962] = {X 326.3622, Y 6.9097, Z -2.1667, A 0.000, B 0.000, C 0.000 }
gfCNCPoint1[24963] = {X 326.7602, Y 6.1106, Z -2.1667, A 0.000, B 0.000, C 0.000 }
gfCNCPoint1[24964] = {X 327.3112, Y 5.4083, Z -2.1667, A 0.000, B 0.000, C 0.000 }
gfCNCPoint1[24965] = {X 327.9926, Y 4.8317, Z -2.1667, A 0.000, B 0.000, C 0.000 }
gfCNCPoint1[24966] = {X 328.6647, Y 4.3715, Z -2.1667, A 0.000, B 0.000, C 0.000 }
gfCNCPoint1[24967] = {X 329.5527, Y 3.9110, Z -2.1667, A 0.000, B 0.000, C 0.000 }
gfCNCPoint1[24968] = {X 330.5217, Y 3.6630, Z -2.1667, A 0.000, B 0.000, C 0.000 }
gfCNCPoint1[24969] = {X 331.5217, Y 3.6402, Z -2.1667, A 0.000, B 0.000, C 0.000 }
gfCNCPoint1[24970] = {X 332.5010, Y 3.8439, Z -2.1667, A 0.000, B 0.000, C 0.000 }
gfCNCPoint1[24971] = {X 333.5113, Y 3.2691, Z -2.1667, A 0.000, B 0.000, C 0.000 }
gfCNCPoint1[24972] = {X 334.5442, Y 2.7360, Z -2.1667, A 0.000, B 0.000, C 0.000 }
gfCNCPoint1[24973] = {X 334.3328, Y 2.3051, Z -2.1667, A 0.000, B 0.000, C 0.000 }
gfCNCPoint1[24974] = {X 2.3035, Y 2.3051, Z -2.1667, A 0.000, B 0.000, C 0.000 }
gfCNCPoint1[24975] = {X 2.3035, Y 6.8598, Z -2.1667, A 0.000, B 0.000, C 0.000 }
gfCNCPoint1[24976] = {X 2.4142, Y 6.8819, Z -2.1667, A 0.000, B 0.000, C 0.000 }
gfCNCPoint1[24977] = {X 2.8632, Y 6.6970, Z -2.1667, A 0.000, B 0.000, C 0.000 }
gfCNCPoint1[24978] = {X 3.3174, Y 6.5253, Z -2.1667, A 0.000, B 0.000, C 0.000 }
gfCNCPoint1[24979] = {X 5.4246, Y 5.7917, Z -2.1667, A 0.000, B 0.000, C 0.000 }
gfCNCPoint1[24980] = {X 7.5870, Y 5.2418, Z -2.1667, A 0.000, B 0.000, C 0.000 }
gfCNCPoint1[24981] = {X 9.7886, Y 4.8797, Z -2.1667, A 0.000, B 0.000, C 0.000 }
gfCNCPoint1[24982] = {X 12.0132, Y 4.7081, Z -2.1667, A 0.000, B 0.000, C 0.000 }
gfCNCPoint1[24983] = {X 14.2444, Y 4.7282, Z -2.1667, A 0.000, B 0.000, C 0.000 }
gfCNCPoint1[24984] = {X 16.4655, Y 4.9400, Z -2.1667, A 0.000, B 0.000, C 0.000 }
gfCNCPoint1[24985] = {X 16.9032, Y 5.0007, Z -2.1667, A 0.000, B 0.000, C 0.000 }
gfCNCPoint1[24986] = {X 17.9958, Y 5.1987, Z -2.1667, A 0.000, B 0.000, C 0.000 }
gfCNCPoint1[24987] = {X 19.0756, Y 5.4572, Z -2.1667, A 0.000, B 0.000, C 0.000 }
gfCNCPoint1[24988] = {X 20.9556, Y 6.0643, Z -2.1667, A 0.000, B 0.000, C 0.000 }
gfCNCPoint1[24989] = {X 22.7662, Y 6.8545, Z -2.1667, A 0.000, B 0.000, C 0.000 }
gfCNCPoint1[24990] = {X 24.4880, Y 7.8189, Z -2.1667, A 0.000, B 0.000, C 0.000 }
gfCNCPoint1[24991] = {X 26.1061, Y 8.9488, Z -2.1667, A 0.000, B 0.000, C 0.000 }
gfCNCPoint1[24992] = {X 27.3995, Y 10.0791, Z -2.1667, A 0.000, B 0.000, C 0.000 }
gfCNCPoint1[24993] = {X 28.5598, Y 11.3455, Z -2.1667, A 0.000, B 0.000, C 0.000 }
gfCNCPoint1[24994] = {X 29.5728, Y 12.7326, Z -2.1667, A 0.000, B 0.000, C 0.000 }
gfCNCPoint1[24995] = {X 30.4262, Y 14.2233, Z -2.1667, A 0.000, B 0.000, C 0.000 }
gfCNCPoint1[24996] = {X 31.1093, Y 15.7992, Z -2.1667, A 0.000, B 0.000, C 0.000 }
gfCNCPoint1[24997] = {X 31.6698, Y 17.7351, Z -2.1667, A 0.000, B 0.000, C 0.000 }
gfCNCPoint1[24998] = {X 32.0035, Y 19.7226, Z -2.1667, A 0.000, B 0.000, C 0.000 }
gfCNCPoint1[24999] = {X 32.1059, Y 21.7353, Z -2.1667, A 0.000, B 0.000, C 0.000 }
gfCNCPoint1[25000] = {X 31.9756, Y 23.7465, Z -2.1667, A 0.000, B 0.000, C 0.000 }
gfCNCPoint1[25001] = {X 31.6143, Y 25.7292, Z -2.1667, A 0.000, B 0.000, C 0.000 }
gfCNCPoint1[25002] = {X 31.1956, Y 27.1579, Z -2.1667, A 0.000, B 0.000, C 0.000 }
gfCNCPoint1[25003] = {X 30.6293, Y 28.5348, Z -2.1667, A 0.000, B 0.000, C 0.000 }
gfCNCPoint1[25004] = {X 29.9216, Y 29.8447, Z -2.1667, A 0.000, B 0.000, C 0.000 }
gfCNCPoint1[25005] = {X 29.0804, Y 31.0731, Z -2.1667, A 0.000, B 0.000, C 0.000 }
gfCNCPoint1[25006] = {X 29.6384, Y 31.7917, Z -2.1667, A 0.000, B 0.000, C 0.000 }
gfCNCPoint1[25007] = {X 30.0954, Y 32.5784, Z -2.1667, A 0.000, B 0.000, C 0.000 }
gfCNCPoint1[25008] = {X 33.1423, Y 38.8726, Z -2.1667, A 0.000, B 0.000, C 0.000 }
gfCNCPoint1[25009] = {X 33.5391, Y 39.8957, Z -2.1667, A 0.000, B 0.000, C 0.000 }
gfCNCPoint1[25010] = {X 33.7662, Y 40.9694, Z -2.1667, A 0.000, B 0.000, C 0.000 }
gfCNCPoint1[25011] = {X 33.8177, Y 42.0656, Z -2.1667, A 0.000, B 0.000, C 0.000 }
gfCNCPoint1[25012] = {X 33.7164, Y 43.0266, Z -2.1667, A 0.000, B 0.000, C 0.000 }
gfCNCPoint1[25013] = {X 33.4799, Y 43.9636, Z -2.1667, A 0.000, B 0.000, C 0.000 }
gfCNCPoint1[25014] = {X 33.1103, Y 44.8630, Z -2.1667, A 0.000, B 0.000, C 0.000 }
gfCNCPoint1[25015] = {X 32.6161, Y 45.7005, Z -2.1667, A 0.000, B 0.000, C 0.000 }
gfCNCPoint1[25016] = {X 32.0075, Y 46.4590, Z -2.1667, A 0.000, B 0.000, C 0.000 }
gfCNCPoint1[25017] = {X 31.2970, Y 47.1229, Z -2.1667, A 0.000, B 0.000, C 0.000 }
gfCNCPoint1[25018] = {X 30.7581, Y 47.5586, Z -2.1667, A 0.000, B 0.000, C 0.000 }
gfCNCPoint1[25019] = {X 29.8522, Y 48.1759, Z -2.1667, A 0.000, B 0.000, C 0.000 }
gfCNCPoint1[25020] = {X 28.8591, Y 48.6401, Z -2.1667, A 0.000, B 0.000, C 0.000 }
gfCNCPoint1[25021] = {X 27.8045, Y 48.9391, Z -2.1667, A 0.000, B 0.000, C 0.000 }
gfCNCPoint1[25022] = {X 26.7155, Y 49.0651, Z -2.1667, A 0.000, B 0.000, C 0.000 }
gfCNCPoint1[25023] = {X 25.6205, Y 49.0151, Z -2.1667, A 0.000, B 0.000, C 0.000 }
gfCNCPoint1[25024] = {X 23.6861, Y 49.9665, Z -2.1667, A 0.000, B 0.000, C 0.000 }
gfCNCPoint1[25025] = {X 21.6902, Y 50.7813, Z -2.1667, A 0.000, B 0.000, C 0.000 }
gfCNCPoint1[25026] = {X 19.6426, Y 51.4553, Z -2.1667, A 0.000, B 0.000, C 0.000 }
gfCNCPoint1[25027] = {X 17.3179, Y 52.0289, Z -2.1667, A 0.000, B 0.000, C 0.000 }
gfCNCPoint1[25028] = {X 14.9491, Y 52.3785, Z -2.1667, A 0.000, B 0.000, C 0.000 }
gfCNCPoint1[25029] = {X 12.5578, Y 52.5009, Z -2.1667, A 0.000, B 0.000, C 0.000 }
gfCNCPoint1[25030] = {X 10.1657, Y 52.3949, Z -2.1667, A 0.000, B 0.000, C 0.000 }
gfCNCPoint1[25031] = {X 7.7946, Y 52.0616, Z -2.1667, A 0.000, B 0.000, C 0.000 }
gfCNCPoint1[25032] = {X 6.6016, Y 51.8039, Z -2.1667, A 0.000, B 0.000, C 0.000 }
gfCNCPoint1[25033] = {X 5.4269, Y 51.4724, Z -2.1667, A 0.000, B 0.000, C 0.000 }
gfCNCPoint1[25034] = {X 3.8373, Y 50.8933, Z -2.1667, A 0.000, B 0.000, C 0.000 }
gfCNCPoint1[25035] = {X 2.3035, Y 50.1792, Z -2.1667, A 0.000, B 0.000, C 0.000 }
gfCNCPoint1[25036] = {X 2.3035, Y 97.6949, Z -2.1667, A 0.000, B 0.000, C 0.000 }
gfCNCPoint1[25037] = {X 120.1200, Y 97.6949, Z -2.1667, A 0.000, B 0.000, C 0.000 }
gfCNCPoint1[25038] = {X 120.1200, Y 97.0659, Z -2.1667, A 0.000, B 0.000, C 0.000 }
gfCNCPoint1[25039] = {X 120.2340, Y 96.0175, Z -2.1667, A 0.000, B 0.000, C 0.000 }
gfCNCPoint1[25040] = {X 120.5705, Y 95.0180, Z -2.1667, A 0.000, B 0.000, C 0.000 }
gfCNCPoint1[25041] = {X 121.1140, Y 94.1141, Z -2.1667, A 0.000, B 0.000, C 0.000 }
gfCNCPoint1[25042] = {X 121.8389, Y 93.3482, Z -2.1667, A 0.000, B 0.000, C 0.000 }
gfCNCPoint1[25043] = {X 122.7115, Y 92.7558, Z -2.1667, A 0.000, B 0.000, C 0.000 }
gfCNCPoint1[25044] = {X 123.6909, Y 92.3648, Z -2.1667, A 0.000, B 0.000, C 0.000 }
gfCNCPoint1[25045] = {X 124.7315, Y 92.1933, Z -2.1667, A 0.000, B 0.000, C 0.000 }
gfCNCPoint1[25046] = {X 124.7883, Y 92.1790, Z -2.1667, A 0.000, B 0.000, C 0.000 }
gfCNCPoint1[25047] = {X 124.8458, Y 92.1685, Z -2.1667, A 0.000, B 0.000, C 0.000 }
gfCNCPoint1[25048] = {X 125.3649, Y 92.0915, Z -2.1667, A 0.000, B 0.000, C 0.000 }
gfCNCPoint1[25049] = {X 126.1001, Y 91.9695, Z -2.1667, A 0.000, B 0.000, C 0.000 }
gfCNCPoint1[25050] = {X 126.8264, Y 91.8024, Z -2.1667, A 0.000, B 0.000, C 0.000 }
gfCNCPoint1[25051] = {X 127.9743, Y 90.7129, Z -2.1667, A 0.000, B 0.000, C 0.000 }
gfCNCPoint1[25052] = {X 129.0639, Y 89.5653, Z -2.1667, A 0.000, B 0.000, C 0.000 }
gfCNCPoint1[25053] = {X 154.9464, Y 61.1428, Z -2.1667, A 0.000, B 0.000, C 0.000 }
gfCNCPoint1[25054] = {X 154.6594, Y 60.4500, Z -2.1667, A 0.000, B 0.000, C 0.000 }
gfCNCPoint1[25055] = {X 154.4819, Y 59.7215, Z -2.1667, A 0.000, B 0.000, C 0.000 }
gfCNCPoint1[25056] = {X 154.4181, Y 58.9744, Z -2.1667, A 0.000, B 0.000, C 0.000 }
gfCNCPoint1[25057] = {X 154.4180, Y 58.0000, Z -2.1667, A 0.000, B 0.000, C 0.000 }
gfCNCPoint1[25058] = {X 154.5117, Y 57.0480, Z -2.1667, A 0.000, B 0.000, C 0.000 }
gfCNCPoint1[25059] = {X 154.7894, Y 56.1325, Z -2.1667, A 0.000, B 0.000, C 0.000 }
gfCNCPoint1[25060] = {X 155.2404, Y 55.2888, Z -2.1667, A 0.000, B 0.000, C 0.000 }
gfCNCPoint1[25061] = {X 155.8473, Y 54.5493, Z -2.1667, A 0.000, B 0.000, C 0.000 }
gfCNCPoint1[25062] = {X 156.5868, Y 53.9424, Z -2.1667, A 0.000, B 0.000, C 0.000 }
gfCNCPoint1[25063] = {X 157.4305, Y 53.4915, Z -2.1667, A 0.000, B 0.000, C 0.000 }
gfCNCPoint1[25064] = {X 158.3459, Y 53.2138, Z -2.1667, A 0.000, B 0.000, C 0.000 }
gfCNCPoint1[25065] = {X 159.2980, Y 53.1200, Z -2.1667, A 0.000, B 0.000, C 0.000 }
gfCNCPoint1[25066] = {X 178.5335, Y 53.1200, Z -2.1667, A 0.000, B 0.000, C 0.000 }
gfCNCPoint1[25067] = {X 179.4855, Y 53.2138, Z -2.1667, A 0.000, B 0.000, C 0.000 }
gfCNCPoint1[25068] = {X 180.4010, Y 53.4915, Z -2.1667, A 0.000, B 0.000, C 0.000 }
gfCNCPoint1[25069] = {X 181.2447, Y 53.9424, Z -2.1667, A 0.000, B 0.000, C 0.000 }
gfCNCPoint1[25070] = {X 181.9842, Y 54.5493, Z -2.1667, A 0.000, B 0.000, C 0.000 }
gfCNCPoint1[25071] = {X 182.5911, Y 55.2888, Z -2.1667, A 0.000, B 0.000, C 0.000 }
gfCNCPoint1[25072] = {X 183.0420, Y 56.1325, Z -2.1667, A 0.000, B 0.000, C 0.000 }
gfCNCPoint1[25073] = {X 183.3197, Y 57.0480, Z -2.1667, A 0.000, B 0.000, C 0.000 }
gfCNCPoint1[25074] = {X 183.4135, Y 58.0000, Z -2.1667, A 0.000, B 0.000, C 0.000 }
gfCNCPoint1[25075] = {X 183.4133, Y 58.9744, Z -2.1667, A 0.000, B 0.000, C 0.000 }
gfCNCPoint1[25076] = {X 183.3512, Y 59.7115, Z -2.1667, A 0.000, B 0.000, C 0.000 }
gfCNCPoint1[25077] = {X 183.1783, Y 60.4308, Z -2.1667, A 0.000, B 0.000, C 0.000 }
gfCNCPoint1[25078] = {X 182.8987, Y 61.1157, Z -2.1667, A 0.000, B 0.000, C 0.000 }
gfCNCPoint1[25079] = {X 209.8904, Y 90.5756, Z -2.1667, A 0.000, B 0.000, C 0.000 }
gfCNCPoint1[25080] = {X 210.5199, Y 91.2142, Z -2.1667, A 0.000, B 0.000, C 0.000 }
gfCNCPoint1[25081] = {X 211.1942, Y 91.8053, Z -2.1667, A 0.000, B 0.000, C 0.000 }
gfCNCPoint1[25082] = {X 211.3600, Y 91.9095, Z -2.1667, A 0.000, B 0.000, C 0.000 }
gfCNCPoint1[25083] = {X 211.5460, Y 91.9703, Z -2.1667, A 0.000, B 0.000, C 0.000 }
gfCNCPoint1[25084] = {X 212.2018, Y 92.1105, Z -2.1667, A 0.000, B 0.000, C 0.000 }
gfCNCPoint1[25085] = {X 213.4082, Y 92.2625, Z -2.1667, A 0.000, B 0.000, C 0.000 }
gfCNCPoint1[25086] = {X 214.4424, Y 92.1762, Z -2.1667, A 0.000, B 0.000, C 0.000 }
gfCNCPoint1[25087] = {X 215.4785, Y 92.1173, Z -2.1667, A 0.000, B 0.000, C 0.000 }
gfCNCPoint1[25088] = {X 216.0525, Y 92.0573, Z -2.1667, A 0.000, B 0.000, C 0.000 }
gfCNCPoint1[25089] = {X 216.6055, Y 91.8919, Z -2.1667, A 0.000, B 0.000, C 0.000 }
gfCNCPoint1[25090] = {X 217.1182, Y 91.6270, Z -2.1667, A 0.000, B 0.000, C 0.000 }
gfCNCPoint1[25091] = {X 244.6020, Y 74.0195, Z -2.1667, A 0.000, B 0.000, C 0.000 }
gfCNCPoint1[25092] = {X 221.4278, Y 64.9248, Z -2.1667, A 0.000, B 0.000, C 0.000 }
gfCNCPoint1[25093] = {X 219.7200, Y 64.3526, Z -2.1667, A 0.000, B 0.000, C 0.000 }
gfCNCPoint1[25094] = {X 217.9579, Y 63.9798, Z -2.1667, A 0.000, B 0.000, C 0.000 }
gfCNCPoint1[25095] = {X 216.1647, Y 63.8112, Z -2.1667, A 0.000, B 0.000, C 0.000 }
gfCNCPoint1[25096] = {X 215.1121, Y 63.6594, Z -2.1667, A 0.000, B 0.000, C 0.000 }
gfCNCPoint1[25097] = {X 214.1174, Y 63.2832, Z -2.1667, A 0.000, B 0.000, C 0.000 }
gfCNCPoint1[25098] = {X 213.2278, Y 62.7005, Z -2.1667, A 0.000, B 0.000, C 0.000 }
gfCNCPoint1[25099] = {X 212.4856, Y 61.9389, Z -2.1667, A 0.000, B 0.000, C 0.000 }
gfCNCPoint1[25100] = {X 211.9260, Y 61.0346, Z -2.1667, A 0.000, B 0.000, C 0.000 }
gfCNCPoint1[25101] = {X 211.5756, Y 60.0305, Z -2.1667, A 0.000, B 0.000, C 0.000 }
gfCNCPoint1[25102] = {X 211.4510, Y 58.9744, Z -2.1667, A 0.000, B 0.000, C 0.000 }
gfCNCPoint1[25103] = {X 211.4508, Y 58.0000, Z -2.1667, A 0.000, B 0.000, C 0.000 }
gfCNCPoint1[25104] = {X 211.5446, Y 57.0480, Z -2.1667, A 0.000, B 0.000, C 0.000 }
gfCNCPoint1[25105] = {X 211.8223, Y 56.1325, Z -2.1667, A 0.000, B 0.000, C 0.000 }
gfCNCPoint1[25106] = {X 212.2732, Y 55.2888, Z -2.1667, A 0.000, B 0.000, C 0.000 }
gfCNCPoint1[25107] = {X 212.8801, Y 54.5493, Z -2.1667, A 0.000, B 0.000, C 0.000 }
gfCNCPoint1[25108] = {X 213.6196, Y 53.9424, Z -2.1667, A 0.000, B 0.000, C 0.000 }
gfCNCPoint1[25109] = {X 214.4633, Y 53.4915, Z -2.1667, A 0.000, B 0.000, C 0.000 }
gfCNCPoint1[25110] = {X 215.3788, Y 53.2138, Z -2.1667, A 0.000, B 0.000, C 0.000 }
gfCNCPoint1[25111] = {X 216.3308, Y 53.1200, Z -2.1667, A 0.000, B 0.000, C 0.000 }
gfCNCPoint1[25112] = {X 237.2617, Y 53.1200, Z -2.1667, A 0.000, B 0.000, C 0.000 }
gfCNCPoint1[25113] = {X 238.3266, Y 53.2376, Z -2.1667, A 0.000, B 0.000, C 0.000 }
gfCNCPoint1[25114] = {X 239.3401, Y 53.5847, Z -2.1667, A 0.000, B 0.000, C 0.000 }
gfCNCPoint1[25115] = {X 240.2535, Y 54.1447, Z -2.1667, A 0.000, B 0.000, C 0.000 }
gfCNCPoint1[25116] = {X 241.0227, Y 54.8905, Z -2.1667, A 0.000, B 0.000, C 0.000 }
gfCNCPoint1[25117] = {X 241.6106, Y 55.7861, Z -2.1667, A 0.000, B 0.000, C 0.000 }
gfCNCPoint1[25118] = {X 241.9889, Y 56.7885, Z -2.1667, A 0.000, B 0.000, C 0.000 }
gfCNCPoint1[25119] = {X 242.1394, Y 57.8492, Z -2.1667, A 0.000, B 0.000, C 0.000 }
gfCNCPoint1[25120] = {X 247.6958, Y 60.0155, Z -2.1667, A 0.000, B 0.000, C 0.000 }
gfCNCPoint1[25121] = {X 275.0737, Y 70.8783, Z -2.1667, A 0.000, B 0.000, C 0.000 }
gfCNCPoint1[25122] = {X 275.0731, Y 63.6743, Z -2.1667, A 0.000, B 0.000, C 0.000 }
gfCNCPoint1[25123] = {X 274.0647, Y 63.3060, Z -2.1667, A 0.000, B 0.000, C 0.000 }
gfCNCPoint1[25124] = {X 273.1612, Y 62.7262, Z -2.1667, A 0.000, B 0.000, C 0.000 }
gfCNCPoint1[25125] = {X 272.4063, Y 61.9628, Z -2.1667, A 0.000, B 0.000, C 0.000 }
gfCNCPoint1[25126] = {X 271.8367, Y 61.0529, Z -2.1667, A 0.000, B 0.000, C 0.000 }
gfCNCPoint1[25127] = {X 271.4798, Y 60.0404, Z -2.1667, A 0.000, B 0.000, C 0.000 }
gfCNCPoint1[25128] = {X 271.3529, Y 58.9744, Z -2.1667, A 0.000, B 0.000, C 0.000 }
gfCNCPoint1[25129] = {X 271.3527, Y 58.0000, Z -2.1667, A 0.000, B 0.000, C 0.000 }
gfCNCPoint1[25130] = {X 271.4465, Y 57.0480, Z -2.1667, A 0.000, B 0.000, C 0.000 }
gfCNCPoint1[25131] = {X 271.7242, Y 56.1325, Z -2.1667, A 0.000, B 0.000, C 0.000 }
gfCNCPoint1[25132] = {X 272.1751, Y 55.2888, Z -2.1667, A 0.000, B 0.000, C 0.000 }
gfCNCPoint1[25133] = {X 272.7820, Y 54.5493, Z -2.1667, A 0.000, B 0.000, C 0.000 }
gfCNCPoint1[25134] = {X 273.5215, Y 53.9424, Z -2.1667, A 0.000, B 0.000, C 0.000 }
gfCNCPoint1[25135] = {X 274.3652, Y 53.4915, Z -2.1667, A 0.000, B 0.000, C 0.000 }
gfCNCPoint1[25136] = {X 275.2806, Y 53.2138, Z -2.1667, A 0.000, B 0.000, C 0.000 }
gfCNCPoint1[25137] = {X 276.2327, Y 53.1200, Z -2.1667, A 0.000, B 0.000, C 0.000 }
gfCNCPoint1[25138] = {X 292.7731, Y 53.1200, Z -2.1667, A 0.000, B 0.000, C 0.000 }
gfCNCPoint1[25139] = {X 293.7251, Y 53.2138, Z -2.1667, A 0.000, B 0.000, C 0.000 }
gfCNCPoint1[25140] = {X 294.6406, Y 53.4915, Z -2.1667, A 0.000, B 0.000, C 0.000 }
gfCNCPoint1[25141] = {X 295.4843, Y 53.9424, Z -2.1667, A 0.000, B 0.000, C 0.000 }
gfCNCPoint1[25142] = {X 296.2238, Y 54.5493, Z -2.1667, A 0.000, B 0.000, C 0.000 }
gfCNCPoint1[25143] = {X 296.8307, Y 55.2888, Z -2.1667, A 0.000, B 0.000, C 0.000 }
gfCNCPoint1[25144] = {X 297.2816, Y 56.1325, Z -2.1667, A 0.000, B 0.000, C 0.000 }
gfCNCPoint1[25145] = {X 297.5593, Y 57.0480, Z -2.1667, A 0.000, B 0.000, C 0.000 }
gfCNCPoint1[25146] = {X 297.6531, Y 58.0000, Z -2.1667, A 0.000, B 0.000, C 0.000 }
gfCNCPoint1[25147] = {X 297.6531, Y 58.9372, Z -2.1667, A 0.000, B 0.000, C 0.000 }
gfCNCPoint1[25148] = {X 297.5305, Y 60.0093, Z -2.1667, A 0.000, B 0.000, C 0.000 }
gfCNCPoint1[25149] = {X 297.1760, Y 61.0286, Z -2.1667, A 0.000, B 0.000, C 0.000 }
gfCNCPoint1[25150] = {X 296.6069, Y 61.9454, Z -2.1667, A 0.000, B 0.000, C 0.000 }
gfCNCPoint1[25151] = {X 295.8508, Y 62.7154, Z -2.1667, A 0.000, B 0.000, C 0.000 }
gfCNCPoint1[25152] = {X 294.9444, Y 63.3010, Z -2.1667, A 0.000, B 0.000, C 0.000 }
gfCNCPoint1[25153] = {X 293.9318, Y 63.6739, Z -2.1667, A 0.000, B 0.000, C 0.000 }
gfCNCPoint1[25154] = {X 293.9318, Y 92.3209, Z -2.1667, A 0.000, B 0.000, C 0.000 }
gfCNCPoint1[25155] = {X 294.9443, Y 92.6964, Z -2.1667, A 0.000, B 0.000, C 0.000 }
gfCNCPoint1[25156] = {X 295.8503, Y 93.2840, Z -2.1667, A 0.000, B 0.000, C 0.000 }
gfCNCPoint1[25157] = {X 296.6061, Y 94.0554, Z -2.1667, A 0.000, B 0.000, C 0.000 }
gfCNCPoint1[25158] = {X 297.1751, Y 94.9733, Z -2.1667, A 0.000, B 0.000, C 0.000 }
gfCNCPoint1[25159] = {X 297.5298, Y 95.9933, Z -2.1667, A 0.000, B 0.000, C 0.000 }
gfCNCPoint1[25160] = {X 297.6531, Y 97.0661, Z -2.1667, A 0.000, B 0.000, C 0.000 }
gfCNCPoint1[25161] = {X 297.6531, Y 97.6949, Z -2.1667, A 0.000, B 0.000, C 0.000 }
gfCNCPoint1[25162] = {X 297.1731, Y 97.6949, Z -2.1667, A 0.000, B 0.000, C 0.000 }
gfCNCPoint1[25163] = {X 297.1731, Y 98.0000, Z -2.1667, A 0.000, B 0.000, C 0.000 }
gfCNCPoint1[25164] = {X 297.0628, Y 98.9791, Z -2.1667, A 0.000, B 0.000, C 0.000 }
gfCNCPoint1[25165] = {X 296.7373, Y 99.9091, Z -2.1667, A 0.000, B 0.000, C 0.000 }
gfCNCPoint1[25166] = {X 296.2131, Y 100.7434, Z -2.1667, A 0.000, B 0.000, C 0.000 }
gfCNCPoint1[25167] = {X 295.5164, Y 101.4401, Z -2.1667, A 0.000, B 0.000, C 0.000 }
gfCNCPoint1[25168] = {X 294.6822, Y 101.9643, Z -2.1667, A 0.000, B 0.000, C 0.000 }
gfCNCPoint1[25169] = {X 293.7522, Y 102.2897, Z -2.1667, A 0.000, B 0.000, C 0.000 }
gfCNCPoint1[25170] = {X 292.7731, Y 102.4000, Z -2.1667, A 0.000, B 0.000, C 0.000 }
gfCNCPoint1[25171] = {X 276.2327, Y 102.4000, Z -2.1667, A 0.000, B 0.000, C 0.000 }
gfCNCPoint1[25172] = {X 275.2536, Y 102.2897, Z -2.1667, A 0.000, B 0.000, C 0.000 }
gfCNCPoint1[25173] = {X 274.3236, Y 101.9643, Z -2.1667, A 0.000, B 0.000, C 0.000 }
gfCNCPoint1[25174] = {X 273.4893, Y 101.4401, Z -2.1667, A 0.000, B 0.000, C 0.000 }
gfCNCPoint1[25175] = {X 272.7926, Y 100.7434, Z -2.1667, A 0.000, B 0.000, C 0.000 }
gfCNCPoint1[25176] = {X 272.2684, Y 99.9091, Z -2.1667, A 0.000, B 0.000, C 0.000 }
gfCNCPoint1[25177] = {X 271.9430, Y 98.9791, Z -2.1667, A 0.000, B 0.000, C 0.000 }
gfCNCPoint1[25178] = {X 271.8327, Y 98.0000, Z -2.1667, A 0.000, B 0.000, C 0.000 }
gfCNCPoint1[25179] = {X 271.8329, Y 97.0190, Z -2.1667, A 0.000, B 0.000, C 0.000 }
gfCNCPoint1[25180] = {X 271.9305, Y 96.1432, Z -2.1667, A 0.000, B 0.000, C 0.000 }
gfCNCPoint1[25181] = {X 272.2006, Y 95.3045, Z -2.1667, A 0.000, B 0.000, C 0.000 }
gfCNCPoint1[25182] = {X 272.6325, Y 94.5364, Z -2.1667, A 0.000, B 0.000, C 0.000 }
gfCNCPoint1[25183] = {X 273.2087, Y 93.8698, Z -2.1667, A 0.000, B 0.000, C 0.000 }
gfCNCPoint1[25184] = {X 273.9062, Y 93.3313, Z -2.1667, A 0.000, B 0.000, C 0.000 }
gfCNCPoint1[25185] = {X 274.6970, Y 92.9426, Z -2.1667, A 0.000, B 0.000, C 0.000 }
gfCNCPoint1[25186] = {X 275.5494, Y 92.7193, Z -2.1667, A 0.000, B 0.000, C 0.000 }
gfCNCPoint1[25187] = {X 275.5494, Y 85.6495, Z -2.1667, A 0.000, B 0.000, C 0.000 }
gfCNCPoint1[25188] = {X 262.6479, Y 80.5921, Z -2.1667, A 0.000, B 0.000, C 0.000 }
gfCNCPoint1[25189] = {X 262.3189, Y 80.7991, Z -2.1667, A 0.000, B 0.000, C 0.000 }
gfCNCPoint1[25190] = {X 237.8763, Y 96.6312, Z -2.1667, A 0.000, B 0.000, C 0.000 }
gfCNCPoint1[25191] = {X 237.8798, Y 97.0659, Z -2.1667, A 0.000, B 0.000, C 0.000 }
gfCNCPoint1[25192] = {X 237.8798, Y 98.0000, Z -2.1667, A 0.000, B 0.000, C 0.000 }
gfCNCPoint1[25193] = {X 237.7695, Y 98.9791, Z -2.1667, A 0.000, B 0.000, C 0.000 }
gfCNCPoint1[25194] = {X 237.4440, Y 99.9091, Z -2.1667, A 0.000, B 0.000, C 0.000 }
gfCNCPoint1[25195] = {X 236.9198, Y 100.7434, Z -2.1667, A 0.000, B 0.000, C 0.000 }
gfCNCPoint1[25196] = {X 236.2231, Y 101.4401, Z -2.1667, A 0.000, B 0.000, C 0.000 }
gfCNCPoint1[25197] = {X 235.3889, Y 101.9643, Z -2.1667, A 0.000, B 0.000, C 0.000 }
gfCNCPoint1[25198] = {X 234.4589, Y 102.2897, Z -2.1667, A 0.000, B 0.000, C 0.000 }
gfCNCPoint1[25199] = {X 233.4798, Y 102.4000, Z -2.1667, A 0.000, B 0.000, C 0.000 }
gfCNCPoint1[25200] = {X 214.1790, Y 102.4000, Z -2.1667, A 0.000, B 0.000, C 0.000 }
gfCNCPoint1[25201] = {X 213.7862, Y 102.3824, Z -2.1667, A 0.000, B 0.000, C 0.000 }
gfCNCPoint1[25202] = {X 213.3966, Y 102.3299, Z -2.1667, A 0.000, B 0.000, C 0.000 }
gfCNCPoint1[25203] = {X 213.0069, Y 102.3824, Z -2.1667, A 0.000, B 0.000, C 0.000 }
